// TwinCAT 3 PLC project PRG_MC_HMI_Conn
// Title: B_MachineControl_HMI_Connector
// Company: RafalOS
// Author: Rafal Osajda
// ProjectVersion: 0.0.0.38
// ProgramVersion: 3.1.4024.0
// libraries:
//   B_Base, * (RafalOS)
//   B_Base_HMI_Connector, * (RafalOS)
//   B_HMIElements, * (RafalOS)
//   B_MachineControl, * (RafalOS)
//   B_StatesAndModes, * (RafalOS)
//   VisuElemBase, * (System)
//   Tc2_Standard, * (Beckhoff Automation GmbH)
//   Tc2_System, * (Beckhoff Automation GmbH)
//   Tc3_Module, * (Beckhoff Automation GmbH)
//   VisuSymbols,3.5.10.0,System
// project tree:
//   DUTs/ ST_MCHMIPrepareScreen_List.TcDUT, ST_MCHMIPrepareScreen_DescriptorList.TcDUT
//   GVLs/ GVL_MCHMIConstans.TcGVL
//   / PlcTask.TcTTO (not stored)
//   POUs Compilation/ PRGCompilation.TcPOU
//   POUs/01_MC/ FB_MCHMIMachineControl_HMI.TcPOU, ITF_MCHMIMachineControl_HMI.TcIO, ITF_MCHMIMachineControl_HMI_PrepScr.TcIO, ITF_MCHMIMachineControl_HMI_PrepScr_00_01.TcIO, ITF_MCHMIMachineControl_HMI_PrepScr_00_02.TcIO, ITF_MCHMIMachineControl_HMI_PrepScr_00_03.TcIO, ITF_MCHMIMachineControl_HMI_PrepScr_00_04.TcIO, ITF_MCHMIMachineControl_HMI_PrepScr_00_05.TcIO, ITF_MCHMIMachineControl_HMI_PrepScr_01_XX.TcIO, ITF_MCHMIMachineControl_HMI_PrepScr_02_XX.TcIO, ITF_MCHMIMachineControl_HMI_PrepScr_03_XX.TcIO, ITF_MCHMIMachineControl_HMI_PrepScr_04_XX.TcIO, ITF_MCHMIMachineControl_HMI_PrepScr_05_XX.TcIO, ITF_MCHMIMachineControl_HMI_PrepScr_06_XX.TcIO, ITF_MCHMIMachineControl_HMI_PrepScr_07_XX.TcIO, ST_MCHMICommonData.TcDUT, ST_MCHMICommonData_RecipeInfo.TcDUT, ST_MCHMIMachineControl_HMI_Link.TcDUT, ST_MCHMIMachineControl_HMI.TcDUT
//   POUs/02_PrepareScreenParent/ FB_MCHMIPrepareDataForScreen.TcPOU, ITF_MCHMIDisplayExtension.TcIO, ITF_MCHMIPrepareDataForScreen.TcIO, ITF_MCHMIPrepareDataForScreenExtension.TcIO, ITF_MCHMIPrepareScreen_Init.TcIO
//   POUs/03_MW_Production/ FB_MCHMIPrepareDataForScreen_00_01.TcPOU, ITF_MCHMIPrepareScreen_00_01_Init.TcIO, ST_MCHMIPrepareScreen_00_01.TcDUT
//   POUs/04_MW_Maitenance/ FB_MCHMIPrepareDataForScreen_00_02.TcPOU, ITF_MCHMIPrepareScreen_00_02_Init.TcIO, ST_MCHMIPrepareScreen_00_02.TcDUT
//   POUs/05_MW_Manual/ FB_MCHMIPrepareDataForScreen_00_03.TcPOU, ITF_MCHMIPrepareScreen_00_03_Init.TcIO, ST_MCHMIPrepareScreen_00_03.TcDUT
//   POUs/06_MW_Washing/ FB_MCHMIPrepareDataForScreen_00_04.TcPOU, ITF_MCHMIPrepareScreen_00_04_Init.TcIO, ST_MCHMIPrepareScreen_00_04.TcDUT
//   POUs/07_MW_Diagnostics/ FB_MCHMIPrepareDataForScreen_00_05.TcPOU, ITF_MCHMIPrepareScreen_00_05_Init.TcIO, ST_MCHMIPrepareScreen_00_05.TcDUT
//   POUs/08_Parameters/ FB_MCHMIPrepareDataForScreen_01_XX.TcPOU, ITF_MCHMIPrepareScreen_01_XX_Init.TcIO, ST_MCHMIPrepareScreen_01_XX.TcDUT, ST_MCHMIPrepareScreen_01_XX_ElementList.TcDUT
//   POUs/09_Recipe/ FB_MCHMIPrepareDataForScreen_02_XX.TcPOU, ITF_MCHMIPrepareScreen_02_XX_Init.TcIO, ST_MCHMIPrepareScreen_02_XX.TcDUT, ST_MCHMIPrepareScreen_02_XX_AddRecipe.TcDUT, ST_MCHMIPrepareScreen_02_XX_DeleteRecipe.TcDUT
//   POUs/10_Alarm/ FB_MCHMIPrepareDataForScreen_03_XX.TcPOU, ITF_MCHMIPrepareScreen_03_XX_Init.TcIO, ST_MCHMIPrepareScreen_03_XX.TcDUT
//   POUs/11_ChangeMode/ FB_MCHMIPrepareDataForScreen_04_XX.TcPOU, ITF_MCHMIPrepareScreen_04_XX_Init.TcIO, ST_MCHMIPrepareScreen_04_XX.TcDUT
//   POUs/12_Statistics/ FB_MCHMIPrepareDataForScreen_05_XX.TcPOU, ITF_MCHMIPrepareScreen_05_XX_Init.TcIO, ST_MCHMIPrepareScreen_05_XX.TcDUT
//   POUs/13_StateDiagram/ FB_MCHMIPrepareDataForScreen_06_XX.TcPOU, ITF_MCHMIPrepareScreen_06_XX_Init.TcIO, ST_MCHMIPrepareScreen_06_XX.TcDUT, ST_MCHMIPrepareScreen_06_XX_ChangeMode.TcDUT, ST_MCHMIPrepareScreen_06_XX_CmdChangeState.TcDUT, ST_MCHMIPrepareScreen_06_XX_State.TcDUT
//   POUs/14_Setings/ FB_MCHMIPrepareDataForScreen_07_XX.TcPOU, ITF_MCHMIPrepareScreen_07_XX_Init.TcIO, ST_MCHMIPrepareScreen_07_XX.TcDUT
//   VISUs/ VisualizationManager.TcVMO (not stored)
// real-time tasks:
//   TASK PlcTask: cycle T#10ms, priority 20, ADS port 350

// ---- DUTs/ST_MCHMIPrepareScreen_List.TcDUT
TYPE ST_MCHMIPrepareScreen_List :
STRUCT
	arrRow					: ARRAY [1..GVL_MCHMIConstans.NUMBER_INDEGRIEND_ON_PAGE] OF ST_BaseHMIDescriptor;
	iSelectedRow			: INT; //numer wybranego składnika
	iSelectedRowPrev		: INT; //numer wybranego składnika - poprzedni
	bSelectedRow			: BOOL;
	
END_STRUCT
END_TYPE

// ---- DUTs/ST_MCHMIPrepareScreen_DescriptorList.TcDUT
TYPE ST_MCHMIPrepareScreen_DescriptorList :
STRUCT
	iTotal				: INT; //całkowita liczba danych do wyświetlenia
	iStartIndex			: INT; //liczba startowa
	iNumberRowOnPage	: INT; //liczbna wierszy na stronie
	iNumberOfPage		: INT; //ilosc stron potrzebnych do wyświetlenia wszystkich danych
	iActualPage			: INT; //aktualna strona
	iPreviewPage		: INT; //Poprzednia strona
	stChossenRow		: ST_BaseHMIDescriptorEdit;
	stList				: ST_MCHMIPrepareScreen_List;
	bRefresh			: BOOL;
END_STRUCT
END_TYPE

// ---- POUs/01_MC/ST_MCHMICommonData.TcDUT
TYPE ST_MCHMICommonData :
STRUCT
	bChangePage				: BOOL; //zmiana strony menu głównego
	wsActualState			: WSTRING;
	wsActualMode			: WSTRING;
	stRecipeInformation		: ST_MCHMICommonData_RecipeInfo;
END_STRUCT
END_TYPE

// ---- POUs/01_MC/ST_MCHMICommonData_RecipeInfo.TcDUT
TYPE ST_MCHMICommonData_RecipeInfo :
STRUCT
	bRecipeSelected			: BOOL;
	wsRecipeInformation		: WSTRING;
	dwBackgroud				: DWORD;
	dwText					: DWORD;
	(* rozpisane tło
	16#<TT><RR><GG><BB>
	<TT> 00-FF Transpoarency
	<RR> 00-FF red
	<GG> 00-FF green
	<BB> 00-FF blue
	*)
	bNewSelectedRecipe		: BOOL;
END_STRUCT
END_TYPE

// ---- POUs/01_MC/ST_MCHMIMachineControl_HMI_Link.TcDUT
TYPE ST_MCHMIMachineControl_HMI_Link EXTENDS ST_BaseTopElement_HMI_Link :
STRUCT
	stMachineControl		: ST_MCHMIMachineControl_HMI;
	stCommonData			: ST_MCHMICommonData;
	stPrepScr_00_01			: ST_MCHMIPrepareScreen_00_01;
	stPrepScr_00_02			: ST_MCHMIPrepareScreen_00_02;
	stPrepScr_00_03			: ST_MCHMIPrepareScreen_00_03;
	stPrepScr_00_04			: ST_MCHMIPrepareScreen_00_04;
	stPrepScr_00_05			: ST_MCHMIPrepareScreen_00_05;
	stPrepScr_01_XX			: ST_MCHMIPrepareScreen_01_XX;
	stPrepScr_02_XX			: ST_MCHMIPrepareScreen_02_XX;
	stPrepScr_03_XX			: ST_MCHMIPrepareScreen_03_XX;
	stPrepScr_04_XX			: ST_MCHMIPrepareScreen_04_XX;
	stPrepScr_05_XX			: ST_MCHMIPrepareScreen_05_XX;
	stPrepScr_06_XX			: ST_MCHMIPrepareScreen_06_XX;
	stPrepScr_07_XX			: ST_MCHMIPrepareScreen_07_XX;
	stRecipe				: ST_BaseRecipe_HMI;
END_STRUCT
END_TYPE

// ---- POUs/01_MC/ST_MCHMIMachineControl_HMI.TcDUT
TYPE ST_MCHMIMachineControl_HMI :
STRUCT
	bZmienna : BOOL;
END_STRUCT
END_TYPE

// ---- POUs/03_MW_Production/ST_MCHMIPrepareScreen_00_01.TcDUT
TYPE ST_MCHMIPrepareScreen_00_01 :
STRUCT
	btmpValue_00_01	: BOOL;
END_STRUCT
END_TYPE

// ---- POUs/04_MW_Maitenance/ST_MCHMIPrepareScreen_00_02.TcDUT
TYPE ST_MCHMIPrepareScreen_00_02 :
STRUCT
	btmpValue_00_02	: BOOL;
END_STRUCT
END_TYPE

// ---- POUs/05_MW_Manual/ST_MCHMIPrepareScreen_00_03.TcDUT
TYPE ST_MCHMIPrepareScreen_00_03 :
STRUCT
	btmpValue_00_03	: BOOL;
END_STRUCT
END_TYPE

// ---- POUs/06_MW_Washing/ST_MCHMIPrepareScreen_00_04.TcDUT
TYPE ST_MCHMIPrepareScreen_00_04 :
STRUCT
	btmpValue_00_04	: BOOL;
END_STRUCT
END_TYPE

// ---- POUs/07_MW_Diagnostics/ST_MCHMIPrepareScreen_00_05.TcDUT
TYPE ST_MCHMIPrepareScreen_00_05 :
STRUCT
	btmpValue_00_05	: BOOL;
END_STRUCT
END_TYPE

// ---- POUs/08_Parameters/ST_MCHMIPrepareScreen_01_XX.TcDUT
TYPE ST_MCHMIPrepareScreen_01_XX :
STRUCT
	stListElement			: ST_MCHMIPrepareScreen_01_XX_ElementList;
	
END_STRUCT
END_TYPE

// ---- POUs/08_Parameters/ST_MCHMIPrepareScreen_01_XX_ElementList.TcDUT
TYPE ST_MCHMIPrepareScreen_01_XX_ElementList :
STRUCT
	arrNames 			: ARRAY  [1..GVL_BaseConstans.MAX_NUMBER_OF_ALL_ITEM] OF WSTRING;
	arrID				: ARRAY  [1..GVL_BaseConstans.MAX_NUMBER_OF_ALL_ITEM] OF UINT;
	iNumber				: INT;	//liczba elementów z parametrami
	itfElement			: ITF_BaseComponent_HMI;	//interfejs wybranego elementu
END_STRUCT
END_TYPE

// ---- POUs/09_Recipe/ST_MCHMIPrepareScreen_02_XX.TcDUT
TYPE ST_MCHMIPrepareScreen_02_XX :
STRUCT
	bRefreshList		: BOOL;	//odświerzenie listy po zmianie listy receptur
	arrNameListRecipe	: ARRAY [1..GVL_BaseConstans.MAX_NUMBER_OF_RECIPES] OF WSTRING;
	arrNameListTemplate	: ARRAY [1..GVL_BaseConstans.MAX_NUMBER_OF_RECIPES] OF WSTRING;
	iNumberOfRecipe		: INT;
	iNumberOfTemplate	: INT;
	iSelectedNameRow	: INT;
	iSelectedNameRowPrev 	: INT; //poprzedni wiersz listy receptur
	bSelectedNameRow	: BOOL;
(*	Wyświetlanie składników	*)
	stIngredientList	: ST_MCHMIPrepareScreen_DescriptorList;
	
(*	Widoczność przycisków	*)
	bVisibleButtonAddFromTemplate	: BOOL;
	bVisibleButtonAddFromRecipe		: BOOL;
	bVisibleButtonDelete			: BOOL;
	bVsibleButtonEditIngredient		: BOOL;
	bVisibleButtonChoose			: BOOL;
	
(*	Tworzenie nowej receptury	- ramka	*)
	stAddRecipe			: ST_MCHMIPrepareScreen_02_XX_AddRecipe;
(*	Ususwanie receptury	*)
	stDeleteRecipe		: ST_MCHMIPrepareScreen_02_XX_DeleteRecipe;
(*	Wybieranie receptury	*)
	bSelectRecipe		: BOOL;
	
END_STRUCT
END_TYPE

// ---- POUs/09_Recipe/ST_MCHMIPrepareScreen_02_XX_AddRecipe.TcDUT
TYPE ST_MCHMIPrepareScreen_02_XX_AddRecipe :
STRUCT
	bNewRecipeFromTemplate	: BOOL;
	bNewRecipeFromRecipe	: BOOL;
	arrListOfName			: ARRAY [1..GVL_BaseConstans.MAX_NUMBER_OF_RECIPES ] OF WSTRING;
	iNumberOfNames			: INT;
	iSelectedName			: INT;
	bSelectedRow			: BOOL;
	stNewNames				: ST_BaseLabel;	//nazwa nowej receptury
	bOk						: BOOL;
	bCancel					: BOOL;	
	wsTitle					: WSTRING;
	wsSource				: WSTRING;
END_STRUCT
END_TYPE

// ---- POUs/09_Recipe/ST_MCHMIPrepareScreen_02_XX_DeleteRecipe.TcDUT
TYPE ST_MCHMIPrepareScreen_02_XX_DeleteRecipe :
STRUCT
	bDeleteRecipe		: BOOL;
	bOK					: BOOL;
	bCancel				: BOOL;
	wsDescription		: WSTRING;
	wsNameRecipe		: WSTRING;
	
END_STRUCT
END_TYPE

// ---- POUs/10_Alarm/ST_MCHMIPrepareScreen_03_XX.TcDUT
TYPE ST_MCHMIPrepareScreen_03_XX :
STRUCT
	btmpValue_03_XX	: BOOL;
END_STRUCT
END_TYPE

// ---- POUs/11_ChangeMode/ST_MCHMIPrepareScreen_04_XX.TcDUT
TYPE ST_MCHMIPrepareScreen_04_XX :
STRUCT
	wsActualMode			: WSTRING;
	eActualMode				: E_BaseMachineMode;
	
	bChangeMode				: BOOL;	//zmien tryb polecenie z HMi
	iSelectedMode			: INT;
	iNumberModeToDisplay	: INT;
	arrNamesOfMode			: ARRAY [0..GVL_SaMConstans.NUMBER_OF_MODES] OF ST_MCHMIPrepareScreen_06_XX_ChangeMode;
	bSelectedRow			: BOOL;
END_STRUCT
END_TYPE

// ---- POUs/12_Statistics/ST_MCHMIPrepareScreen_05_XX.TcDUT
TYPE ST_MCHMIPrepareScreen_05_XX :
STRUCT
	btmpValue_05_XX	: BOOL;
END_STRUCT
END_TYPE

// ---- POUs/13_StateDiagram/ST_MCHMIPrepareScreen_06_XX.TcDUT
TYPE ST_MCHMIPrepareScreen_06_XX :
STRUCT
	wsActualState			: WSTRING;
	wsActualMode			: WSTRING;
	eActualMode				: E_BaseMachineMode;
	(*	Informacje o stanach w trybie	*)
	arrState				: ARRAY [0..GVL_SaMConstans.NUMBER_OF_STATES] OF ST_MCHMIPrepareScreen_06_XX_State;
	arrStateEnabledInMode	: ARRAY [0..GVL_SaMConstans.NUMBER_OF_STATES] OF BOOL;
	(*	Dane dotyczące wyświetlania czasów 	*)
	bShowTime				: BOOL;
	sTotalWorkTime			: STRING;
	iNumberModeToShowTime	: INT;
	sWorkingTimeInMode		: STRING;
	sNameOfModeShown		: STRING;	//nazwa trybu pokazywanego trybu
	bNextModeToDisplayTime	: BOOL;
	bPrevModeToDisplayTime	: BOOL;
	wsNameModeOfTimeDisplay	: WSTRING;

	
	(*	Przyciski poleceń zmiany stany	*)
	arrCmdChangeState		: ARRAY [1..GVL_SaMConstans.NUMBER_OF_COMMAND_CHANGE_STATES] OF ST_MCHMIPrepareScreen_06_XX_CmdChangeState;

	(*	Obsługa zmiany trybu	*)
	bChangeMode				: BOOL;	//zmien tryb polecenie z HMi
	iSelectedMode			: INT;
	iNumberModeToDisplay	: INT;
	arrNamesOfMode			: ARRAY [0..GVL_SaMConstans.NUMBER_OF_MODES] OF ST_MCHMIPrepareScreen_06_XX_ChangeMode;
	bSelectedRow			: BOOL;
END_STRUCT
END_TYPE

// ---- POUs/13_StateDiagram/ST_MCHMIPrepareScreen_06_XX_ChangeMode.TcDUT
TYPE ST_MCHMIPrepareScreen_06_XX_ChangeMode :
STRUCT
	wsDescription			: WSTRING;
	iNumber					: INT;	//numer trybu
END_STRUCT
END_TYPE

// ---- POUs/13_StateDiagram/ST_MCHMIPrepareScreen_06_XX_CmdChangeState.TcDUT
TYPE ST_MCHMIPrepareScreen_06_XX_CmdChangeState :
STRUCT
	bPushed		: BOOL;
	bEnabled	: BOOL;
END_STRUCT
END_TYPE

// ---- POUs/13_StateDiagram/ST_MCHMIPrepareScreen_06_XX_State.TcDUT
TYPE ST_MCHMIPrepareScreen_06_XX_State :
STRUCT
	wsNameOfState			: WSTRING;
	iWidthFrame				: INT := 1;
	bShowTime				: BOOL;
	sTime					: STRING;
	dwBackgroud				: DWORD;
	(* rozpisane tło
	16#<TT><RR><GG><BB>
	<TT> 00-FF Transpoarency
	<RR> 00-FF red
	<GG> 00-FF green
	<BB> 00-FF blue
	*)
END_STRUCT
END_TYPE

// ---- POUs/14_Setings/ST_MCHMIPrepareScreen_07_XX.TcDUT
TYPE ST_MCHMIPrepareScreen_07_XX :
STRUCT
	arrLocationDescription	: ARRAY  [0..GVL_BaseConstans.NUMBER_OF_LOCATIONS] OF WSTRING;
	iChoosoLocation			: INT;
	
	bCreateRecipeTemplate 	: BOOL;
END_STRUCT
END_TYPE

// ---- GVLs/GVL_MCHMIConstans.TcGVL
{attribute 'qualified_only'}
VAR_GLOBAL CONSTANT
	NUMBER_INDEGRIEND_ON_PAGE	: INT := 10;	//liczba wyświetlanych składników recepury w trybie domyślnym
	
END_VAR

// ---- POUs/01_MC/ITF_MCHMIMachineControl_HMI.TcIO
(*			
	RafalOS
	Rafał Osajda		20.11.2025		TC 4024.66
	Interfejs umożliwający wywoływanie moted z HMIManager
*)
INTERFACE ITF_MCHMIMachineControl_HMI EXTENDS ITF_BaseTopElement_HMI

METHOD PUBLIC AddPrepareScreenModuleFromManager : BOOL
VAR_INPUT
	itfModule	: ITF_MCHMIPrepareScreen_Init;// ITF_MCHMIPrepareDataForScreen;
END_VAR
END_METHOD

(*			
	RafalOS
	Rafał Osajda		26.11.2025		TC 4024.66
	Podłaczenie modułu receptur
*)
METHOD PUBLIC AddRecipeModulFormManager : BOOL
VAR_INPUT
	fbRecipeModul		: ITF_BaseRecipe_HMI;
END_VAR
END_METHOD

(*			
	RafalOS
	Rafał Osajda		19.11.2025		TC 4024.66
	Sprzątanie po stronie wywoływane z HMIManager i wywołująca odpowiednią metode z ITF z arrPrepareScreen
*)
METHOD ClearAfterScreenFroHMIManager : BOOL
VAR_INPUT
	iScreen		: INT;
	iMode		: INT;
END_VAR
END_METHOD

METHOD PUBLIC GetActiveModeFromManager : E_BaseMachineMode
VAR_INPUT
END_VAR
END_METHOD

(*			
	RafalOS
	Rafał Osajda		07.12.2025		TC 4024.66
	Pobierz informacje o aktualnym stanie recepur tzn o tym czy jest wybrana a jak tak to która
*)
METHOD PUBLIC GetInformationLatestRecipes
VAR_INPUT
END_VAR
END_METHOD

METHOD PUBLIC LinkMachineControlData : BOOL
VAR_INPUT
	stData			: REFERENCE TO ST_MCHMIMachineControl_HMI_Link;
END_VAR
END_METHOD

(*			
	RafalOS
	Rafał Osajda		20.11.2025		TC 4024.66
	Podpięcie modułu generowania danych do odpowiedniej pozycji w tablicy [Okno][Tryb]
*)
METHOD PUBLIC LinkPrepareScreenToArrayFromConfiguration : BOOL
VAR_INPUT
	iScreen		: INT;
	iMode		: INT;
	itfModule	: ITF_MCHMIPrepareDataForScreen;
END_VAR
END_METHOD

(*			
	RafalOS
	Rafał Osajda		19.11.2025		TC 4024.66
	Przygotowanie danych dla strony wywoływane z HMIManager i wywołująca odpowiednią metode z ITF z arrPrepareScreen
*)
METHOD PrepareDataForScreenFromHMIManager : BOOL
VAR_INPUT
	iScreen		: INT;
	iMode		: INT;
END_VAR
END_METHOD

(*			
	RafalOS
	Rafał Osajda		19.11.2025		TC 4024.66
	Przygotowanie strony wywoływane z HMIManager i wywołująca odpowiednią metode z ITF z arrPrepareScreen
*)
METHOD PrepareForScreenFromHMIManager : BOOL
VAR_INPUT
	iScreen		: INT;
	iMode		: INT;
END_VAR
END_METHOD

(*			
	RafalOS
	Rafał Osajda		20.11.2025		TC 4024.66
	Ustawienei zmiennej w wspólnych zmiennych z managera
*)
METHOD PUBLIC SetChangePageFromManager : BOOL
VAR_INPUT
	bValue	: BOOL;
END_VAR
END_METHOD

END_INTERFACE

// ---- POUs/01_MC/ITF_MCHMIMachineControl_HMI_PrepScr.TcIO
INTERFACE ITF_MCHMIMachineControl_HMI_PrepScr EXTENDS ITF_MCHMIMachineControl_HMI_PrepScr_00_01, 
	ITF_MCHMIMachineControl_HMI_PrepScr_00_02,
	ITF_MCHMIMachineControl_HMI_PrepScr_00_03,
	ITF_MCHMIMachineControl_HMI_PrepScr_00_04,
	ITF_MCHMIMachineControl_HMI_PrepScr_00_05,
	ITF_MCHMIMachineControl_HMI_PrepScr_01_XX,
	ITF_MCHMIMachineControl_HMI_PrepScr_02_XX,
	ITF_MCHMIMachineControl_HMI_PrepScr_03_XX,
	ITF_MCHMIMachineControl_HMI_PrepScr_04_XX,
	ITF_MCHMIMachineControl_HMI_PrepScr_05_XX,
	ITF_MCHMIMachineControl_HMI_PrepScr_06_XX,
	ITF_MCHMIMachineControl_HMI_PrepScr_07_XX

END_INTERFACE

// ---- POUs/01_MC/ITF_MCHMIMachineControl_HMI_PrepScr_00_01.TcIO
(*			
	RafalOS
	Rafał Osajda		20.11.2025		TC 4024.66
	Interfejs przekazywany do modułów tworzących strony
*)
INTERFACE ITF_MCHMIMachineControl_HMI_PrepScr_00_01

END_INTERFACE

// ---- POUs/01_MC/ITF_MCHMIMachineControl_HMI_PrepScr_00_02.TcIO
(*			
	RafalOS
	Rafał Osajda		20.11.2025		TC 4024.66
	Interfejs przekazywany do modułów tworzących strony
*)
INTERFACE ITF_MCHMIMachineControl_HMI_PrepScr_00_02

END_INTERFACE

// ---- POUs/01_MC/ITF_MCHMIMachineControl_HMI_PrepScr_00_03.TcIO
(*			
	RafalOS
	Rafał Osajda		20.11.2025		TC 4024.66
	Interfejs przekazywany do modułów tworzących strony
*)
INTERFACE ITF_MCHMIMachineControl_HMI_PrepScr_00_03

END_INTERFACE

// ---- POUs/01_MC/ITF_MCHMIMachineControl_HMI_PrepScr_00_04.TcIO
(*			
	RafalOS
	Rafał Osajda		20.11.2025		TC 4024.66
	Interfejs przekazywany do modułów tworzących strony
*)
INTERFACE ITF_MCHMIMachineControl_HMI_PrepScr_00_04

END_INTERFACE

// ---- POUs/01_MC/ITF_MCHMIMachineControl_HMI_PrepScr_00_05.TcIO
(*			
	RafalOS
	Rafał Osajda		20.11.2025		TC 4024.66
	Interfejs przekazywany do modułów tworzących strony
*)
INTERFACE ITF_MCHMIMachineControl_HMI_PrepScr_00_05

END_INTERFACE

// ---- POUs/01_MC/ITF_MCHMIMachineControl_HMI_PrepScr_01_XX.TcIO
(*			
	RafalOS
	Rafał Osajda		20.11.2025		TC 4024.66
	Interfejs przekazywany do modułów tworzących strony
*)
INTERFACE ITF_MCHMIMachineControl_HMI_PrepScr_01_XX

(*			
	RafalOS
	Rafał Osajda		17.12.2025		TC 4024.66
	Pobiera listę elementów które posiadaja parametr i 
	przypisuje ja do zadanej struktury i zwraca true jak się uda
*)
METHOD GetElementNamesWithParameter : BOOL
VAR_INPUT
	stDane			: REFERENCE TO ST_MCElementListWithParameter;
END_VAR
END_METHOD

END_INTERFACE

// ---- POUs/01_MC/ITF_MCHMIMachineControl_HMI_PrepScr_02_XX.TcIO
(*			
	RafalOS
	Rafał Osajda		20.11.2025		TC 4024.66
	Interfejs przekazywany do modułów tworzących strony
*)
INTERFACE ITF_MCHMIMachineControl_HMI_PrepScr_02_XX

(*			
	RafalOS
	Rafał Osajda		03.03.2025		TC 4026.13		wer. 0.0.0.1
	Kopiuje składniki z wybranej receptury i tworzy nową recepture
*)
METHOD PUBLIC AddRecipeFromRecipe : BOOL
VAR_INPUT
	uiNumberRecipe				: UINT;
	stTexts						: ST_BaseLabel;
END_VAR
END_METHOD

(*			
	RafalOS
	Rafał Osajda		03.03.2025		TC 4026.13		wer. 0.0.0.1
	Kopiuje składniki z wybranego szablonu i tworzy nową recepture
*)
METHOD PUBLIC AddRecipeFromTemplate : BOOL
VAR_INPUT
	uiNumberTemplates			: UINT;
	stTexts						: ST_BaseLabel;
END_VAR
END_METHOD

(*			
	RafalOS
	Rafał Osajda		03.06.2025		TC 4024.66
	usuwa referencje do wybranej
*)
METHOD PUBLIC ClearChosen
VAR_INPUT
END_VAR
END_METHOD

(*			
	RafalOS
	Rafał Osajda		03.03.2025		TC 4026.13		wer. 0.0.0.1
	
*)
METHOD PUBLIC DeleteRecipe : BOOL
VAR_INPUT
	uiNumber				: uint;
END_VAR
END_METHOD

(*			
	RafalOS
	Rafał Osajda		03.03.2025		TC 4026.13		wer. 0.0.0.1
	
*)
METHOD PUBLIC GetIngredientFromRecipe : ST_BaseDescriptor
VAR_INPUT
	uiNumberOfRecipe			: UINT;
	uiNumberOfIngredient		: UINT;
END_VAR
END_METHOD

(*			
	RafalOS
	Rafał Osajda		02.12.2025		TC 4024.66
	Zwraca do tablicy wybrany zakres składników
*)
METHOD PUBLIC GetIngredientRange 
VAR_INPUT
	iRecipe			: INT;	//numer receptury z której bierzemy składniki
	iStartIndex		: INT;	//numer startowy składnika
	iCount			: INT;	//ilośc pobieranych 
END_VAR
VAR_IN_OUT
	arrOut : ARRAY [*] OF ST_BaseDescriptor;
END_VAR
VAR_OUTPUT
	iNumberOfFilledData	: INT;	//ilosc wypelnionych danych na strone
END_VAR
END_METHOD

METHOD PUBLIC GetListOfNameRecipe : ST_BaseRecipeList
VAR_INPUT
END_VAR
END_METHOD

METHOD PUBLIC GetListOfNameTemplate : ST_BaseRecipeList
VAR_INPUT
END_VAR
END_METHOD

(*			
	RafalOS
	Rafał Osajda		03.03.2025		TC 4026.13		wer. 0.0.0.1
	
*)
METHOD PUBLIC GetNumberIngredientOfRecipe : UINT
VAR_INPUT
	uiNumber				: UINT;
END_VAR
END_METHOD

METHOD PUBLIC GetNumberOfChoosen : UINT
VAR_INPUT
END_VAR
END_METHOD

METHOD PUBLIC GetNumberOfRecipe : UINT
VAR_INPUT
END_VAR
END_METHOD

METHOD PUBLIC GetNumberOfTemplate : UINT
VAR_INPUT
END_VAR
END_METHOD

(*			
	RafalOS
	Rafał Osajda		06.12.2025		TC 4024.66
	Wybranie receputury
*)
METHOD SelectRecipe : BOOL
VAR_INPUT
	uiRecipe: UINT;
END_VAR
END_METHOD

(*			
	RafalOS
	Rafał Osajda		05.12.2025		TC 4024.66
	Ustawia nową wartośc w podanym składniku
*)
METHOD PUBLIC SetIngredientValue
VAR_INPUT
	iRecipe			: int;
	iIngredient		: INT;
	rValue			: REAL;
END_VAR
END_METHOD

END_INTERFACE

// ---- POUs/01_MC/ITF_MCHMIMachineControl_HMI_PrepScr_03_XX.TcIO
(*			
	RafalOS
	Rafał Osajda		20.11.2025		TC 4024.66
	Interfejs przekazywany do modułów tworzących strony
*)
INTERFACE ITF_MCHMIMachineControl_HMI_PrepScr_03_XX

END_INTERFACE

// ---- POUs/01_MC/ITF_MCHMIMachineControl_HMI_PrepScr_04_XX.TcIO
(*			
	RafalOS
	Rafał Osajda		20.11.2025		TC 4024.66
	Interfejs przekazywany do modułów tworzących strony
*)
INTERFACE ITF_MCHMIMachineControl_HMI_PrepScr_04_XX

METHOD GetActiveMode : E_BaseMachineMode
VAR_INPUT
END_VAR
END_METHOD

METHOD PUBLIC GetActiveModeName : ST_BaseLabel
VAR_INPUT
END_VAR
END_METHOD

(*			
	RafalOS
	Rafał Osajda		25.11.2025		TC 4024.66
	Zwraca nazwę trybu o zadanym numerze
*)
METHOD GetModeName : ST_BaseLabel
VAR_INPUT
	iMode	: INT;
END_VAR
END_METHOD

(*			
	RafalOS
	Rafał Osajda		25.11.2025		TC 4024.66
	Zwraca czy tryb o podanym numerze jest włączony
*)
METHOD IsModeEnabled : BOOL
VAR_INPUT
	iMode 	: INT;
END_VAR
END_METHOD

(*			
	RafalOS
	Rafał Osajda		24.11.2025		TC 4024.66
	Zmien tryb
*)
METHOD SetCmdChangeMode : BOOL
VAR_INPUT
	eCmdNumber	: E_SaMCommandChangeMode;
END_VAR
END_METHOD

END_INTERFACE

// ---- POUs/01_MC/ITF_MCHMIMachineControl_HMI_PrepScr_05_XX.TcIO
(*			
	RafalOS
	Rafał Osajda		20.11.2025		TC 4024.66
	Interfejs przekazywany do modułów tworzących strony
*)
INTERFACE ITF_MCHMIMachineControl_HMI_PrepScr_05_XX

END_INTERFACE

// ---- POUs/01_MC/ITF_MCHMIMachineControl_HMI_PrepScr_06_XX.TcIO
(*			
	RafalOS
	Rafał Osajda		20.11.2025		TC 4024.66
	Interfejs przekazywany do modułów tworzących strony
*)
INTERFACE ITF_MCHMIMachineControl_HMI_PrepScr_06_XX

METHOD GetActiveMode : E_BaseMachineMode
VAR_INPUT
END_VAR
END_METHOD

METHOD PUBLIC GetActiveModeName : ST_BaseLabel
VAR_INPUT
END_VAR
END_METHOD

METHOD GetActiveState : E_BaseMachineState
VAR_INPUT
END_VAR
END_METHOD

METHOD PUBLIC GetActiveStateName : ST_BaseLabel
VAR_INPUT
END_VAR
END_METHOD

(*			
	RafalOS
	Rafał Osajda		25.11.2025		TC 4024.66
	Zwraca nazwę trybu o zadanym numerze
*)
METHOD GetModeName : ST_BaseLabel
VAR_INPUT
	iMode	: INT;
END_VAR
END_METHOD

METHOD GetStateName : ST_BaseLabel
VAR_INPUT
	iNumber		: INT;
END_VAR
END_METHOD

METHOD GetStateTimeForMode : LTIME
VAR_INPUT
	iMode		: INT;
	iState		: INT;
END_VAR
END_METHOD

METHOD GetTimeWorkForMode : LTIME
VAR_INPUT
	iMode	: INT;
END_VAR
END_METHOD

(*			
	RafalOS
	Rafał Osajda		25.11.2025		TC 4024.66
	Zwraca całkowity czas pracy maszyny
*)
METHOD PUBLIC GetTotalWorkTime : LTIME
VAR_INPUT
END_VAR
END_METHOD

(*			
	RafalOS
	Rafał Osajda		25.11.2025		TC 4024.66
	Zwraca czy zmiana stanu sie skońćzyła
*)
METHOD IsChangeModeDone : BOOL
VAR_INPUT
END_VAR
END_METHOD

(*			
	RafalOS
	Rafał Osajda		25.11.2025		TC 4024.66
	Zwraca czy tryb o podanym numerze jest włączony
*)
METHOD IsModeEnabled : BOOL
VAR_INPUT
	iMode 	: INT;
END_VAR
END_METHOD

METHOD IsStateActive : BOOL
VAR_INPUT
	iTestState : INT;
END_VAR
END_METHOD

METHOD IsStateEnableInMode : BOOL
VAR_INPUT
	iTestState	: INT;
END_VAR
END_METHOD

(*			
	RafalOS
	Rafał Osajda		24.11.2025		TC 4024.66
	Zmien tryb
*)
METHOD SetCmdChangeMode : BOOL
VAR_INPUT
	eCmdNumber	: E_SaMCommandChangeMode;
END_VAR
END_METHOD

(*			
	RafalOS
	Rafał Osajda		24.11.2025		TC 4024.66
	Zmien stan 
*)
METHOD public SetCmdChangeState : BOOL
VAR_INPUT
	eCmdNumber : E_SaMCommandChangeState;
END_VAR
END_METHOD

END_INTERFACE

// ---- POUs/01_MC/ITF_MCHMIMachineControl_HMI_PrepScr_07_XX.TcIO
(*			
	RafalOS
	Rafał Osajda		20.11.2025		TC 4024.66
	Interfejs przekazywany do modułów tworzących strony
*)
INTERFACE ITF_MCHMIMachineControl_HMI_PrepScr_07_XX

(*			
	RafalOS
	Rafał Osajda		25.10.2025		TC 4024.66
	Utworzenie nowych szablonów receptur na podstawie dodanych fb zewnętrznych - wywołanie metody powoduje
	skosowanie dotychczasowych szablonów i receptur
*)
METHOD PUBLIC CreateRecipeTemplates : BOOL
VAR_INPUT
END_VAR
END_METHOD

END_INTERFACE

// ---- POUs/02_PrepareScreenParent/ITF_MCHMIDisplayExtension.TcIO
INTERFACE ITF_MCHMIDisplayExtension

(*			
	RafalOS
	Rafał Osajda		19.11.2025		TC 4024.66
	Czyści danych przy zmienia ramki po poprzedniej ramce
*)
METHOD PUBLIC ExtendedClearAfterScreen : BOOL
VAR_INPUT
END_VAR
END_METHOD

(*			
	RafalOS
	Rafał Osajda		20.11.2025		TC 4024.66
	Przygotuj rozszerzone wyświetlanie
*)
METHOD PUBLIC ExtendedPrepareDataForHMI : BOOL
VAR_INPUT
END_VAR
END_METHOD

(*			
	RafalOS
	Rafał Osajda		19.11.2025		TC 4024.66
	Przygotowanie ramki pood tamke do wyświetlenia - tylko przygotowanie a nie przygotowanie danych do wyświetlenia
*)
METHOD PUBLIC ExtendedPrepareForScreen : BOOL
VAR_INPUT
END_VAR
END_METHOD

END_INTERFACE

// ---- POUs/02_PrepareScreenParent/ITF_MCHMIPrepareDataForScreen.TcIO
INTERFACE ITF_MCHMIPrepareDataForScreen EXTENDS ITF_BaseComponent_HMI

(*			
	RafalOS
	Rafał Osajda		19.11.2025		TC 4024.66
	Czyści danych przy zmienia ramki po poprzedniej ramce
*)
METHOD PUBLIC ClearAfterScreen : BOOL
VAR_INPUT
END_VAR
END_METHOD

(*			
	RafalOS
	Rafał Osajda		14.11.2025		TC 4024.66
	Metoda przygotowywania danych dla HMI 
	W niej odbywa się odpytywanie właściego elementu przez łącznik
*)
METHOD PUBLIC PrepareDataForHMI : BOOL
VAR_INPUT
END_VAR
END_METHOD

(*			
	RafalOS
	Rafał Osajda		19.11.2025		TC 4024.66
	Przygotowanie ramki pood tamke do wyświetlenia - tylko przygotowanie a nie przygotowanie danych do wyświetlenia
*)
METHOD PUBLIC PrepareForScreen : BOOL
VAR_INPUT
END_VAR
END_METHOD

END_INTERFACE

// ---- POUs/02_PrepareScreenParent/ITF_MCHMIPrepareDataForScreenExtension.TcIO
INTERFACE ITF_MCHMIPrepareDataForScreenExtension

METHOD PUBLIC LinkExtensionDisplay : BOOL
VAR_INPUT
	fbExtendedDisplay			: ITF_MCHMIDisplayExtension;
END_VAR
END_METHOD

END_INTERFACE

// ---- POUs/02_PrepareScreenParent/ITF_MCHMIPrepareScreen_Init.TcIO
INTERFACE ITF_MCHMIPrepareScreen_Init EXTENDS ITF_MCHMIPrepareDataForScreen,
	ITF_MCHMIPrepareScreen_00_01_Init, 
	ITF_MCHMIPrepareScreen_00_02_Init,
	ITF_MCHMIPrepareScreen_00_03_Init,
	ITF_MCHMIPrepareScreen_00_04_Init,
	ITF_MCHMIPrepareScreen_00_05_Init,
	ITF_MCHMIPrepareScreen_01_XX_Init,
	ITF_MCHMIPrepareScreen_02_XX_Init,
	ITF_MCHMIPrepareScreen_03_XX_Init,
	ITF_MCHMIPrepareScreen_04_XX_Init,
	ITF_MCHMIPrepareScreen_05_XX_Init,
	ITF_MCHMIPrepareScreen_06_XX_Init,
	ITF_MCHMIPrepareScreen_07_XX_Init,
	ITF_MCHMIPrepareDataForScreenExtension

(*			
	RafalOS
	Rafał Osajda		20.11.2025		TC 4024.66
	Podłączenie wspólnych danych do modułu 
*)
METHOD PUBLIC LinkHMICommonData : BOOL
VAR_INPUT
	stHMICommonData	: REFERENCE TO ST_MCHMICommonData;
END_VAR
END_METHOD

END_INTERFACE

// ---- POUs/03_MW_Production/ITF_MCHMIPrepareScreen_00_01_Init.TcIO
INTERFACE ITF_MCHMIPrepareScreen_00_01_Init

METHOD PUBLIC LinkDataHMI_00_01 : BOOL
VAR_INPUT
	refstData				: REFERENCE TO ST_MCHMIPrepareScreen_00_01;
END_VAR
END_METHOD

END_INTERFACE

// ---- POUs/04_MW_Maitenance/ITF_MCHMIPrepareScreen_00_02_Init.TcIO
INTERFACE ITF_MCHMIPrepareScreen_00_02_Init

METHOD PUBLIC LinkDataHMI_00_02 : BOOL
VAR_INPUT
	refstData				: REFERENCE TO ST_MCHMIPrepareScreen_00_02;
END_VAR
END_METHOD

END_INTERFACE

// ---- POUs/05_MW_Manual/ITF_MCHMIPrepareScreen_00_03_Init.TcIO
INTERFACE ITF_MCHMIPrepareScreen_00_03_Init

METHOD PUBLIC LinkDataHMI_00_03 : BOOL
VAR_INPUT
	refstData				: REFERENCE TO ST_MCHMIPrepareScreen_00_03;
END_VAR
END_METHOD

END_INTERFACE

// ---- POUs/06_MW_Washing/ITF_MCHMIPrepareScreen_00_04_Init.TcIO
INTERFACE ITF_MCHMIPrepareScreen_00_04_Init

METHOD PUBLIC LinkDataHMI_00_04 : BOOL
VAR_INPUT
	refstData				: REFERENCE TO ST_MCHMIPrepareScreen_00_04;
END_VAR
END_METHOD

END_INTERFACE

// ---- POUs/07_MW_Diagnostics/ITF_MCHMIPrepareScreen_00_05_Init.TcIO
INTERFACE ITF_MCHMIPrepareScreen_00_05_Init

METHOD PUBLIC LinkDataHMI_00_05 : BOOL
VAR_INPUT
	refstData				: REFERENCE TO ST_MCHMIPrepareScreen_00_05;
END_VAR
END_METHOD

END_INTERFACE

// ---- POUs/08_Parameters/ITF_MCHMIPrepareScreen_01_XX_Init.TcIO
INTERFACE ITF_MCHMIPrepareScreen_01_XX_Init

METHOD PUBLIC LinkDataHMI_01_XX : BOOL
VAR_INPUT
	refstData				: REFERENCE TO ST_MCHMIPrepareScreen_01_XX;
END_VAR
END_METHOD

END_INTERFACE

// ---- POUs/09_Recipe/ITF_MCHMIPrepareScreen_02_XX_Init.TcIO
INTERFACE ITF_MCHMIPrepareScreen_02_XX_Init

METHOD PUBLIC LinkDataHMI_02_XX : BOOL
VAR_INPUT
	refstData				: REFERENCE TO ST_MCHMIPrepareScreen_02_XX;
END_VAR
END_METHOD

END_INTERFACE

// ---- POUs/10_Alarm/ITF_MCHMIPrepareScreen_03_XX_Init.TcIO
INTERFACE ITF_MCHMIPrepareScreen_03_XX_Init

METHOD PUBLIC LinkDataHMI_03_XX : BOOL
VAR_INPUT
	refstData				: REFERENCE TO ST_MCHMIPrepareScreen_03_XX;
END_VAR
END_METHOD

END_INTERFACE

// ---- POUs/11_ChangeMode/ITF_MCHMIPrepareScreen_04_XX_Init.TcIO
INTERFACE ITF_MCHMIPrepareScreen_04_XX_Init

METHOD PUBLIC LinkDataHMI_04_XX : BOOL
VAR_INPUT
	refstData				: REFERENCE TO ST_MCHMIPrepareScreen_04_XX;
END_VAR
END_METHOD

END_INTERFACE

// ---- POUs/12_Statistics/ITF_MCHMIPrepareScreen_05_XX_Init.TcIO
INTERFACE ITF_MCHMIPrepareScreen_05_XX_Init

METHOD PUBLIC LinkDataHMI_05_XX : BOOL
VAR_INPUT
	refstData				: REFERENCE TO ST_MCHMIPrepareScreen_05_XX;
END_VAR
END_METHOD

END_INTERFACE

// ---- POUs/13_StateDiagram/ITF_MCHMIPrepareScreen_06_XX_Init.TcIO
INTERFACE ITF_MCHMIPrepareScreen_06_XX_Init

METHOD PUBLIC LinkDataHMI_06_XX : BOOL
VAR_INPUT
	refstData				: REFERENCE TO ST_MCHMIPrepareScreen_06_XX;
END_VAR
END_METHOD

END_INTERFACE

// ---- POUs/14_Setings/ITF_MCHMIPrepareScreen_07_XX_Init.TcIO
INTERFACE ITF_MCHMIPrepareScreen_07_XX_Init

METHOD PUBLIC LinkDataHMI_07_XX : BOOL
VAR_INPUT
	refstData				: REFERENCE TO ST_MCHMIPrepareScreen_07_XX;
END_VAR
END_METHOD

END_INTERFACE

// ---- POUs Compilation/PRGCompilation.TcPOU
PROGRAM PRGCompilation
VAR
	fbLogger						: FB_BaseLogger;
	fbMachineControl				: FB_MCMachineControl;
	fbMachineControlHMIConnector	: FB_MCHMIMachineControl_HMI (
										itfBaseLoggerConnector		:= fbLogger,
	                                    itfMachineControlConnector	:= fbMachineControl
									);
	fbPrepareScreen					: FB_MCHMIPrepareDataForScreen;
	fbPrepareScreen_00_01			: FB_MCHMIPrepareDataForScreen_00_01;
	fbPrepareScreen_00_02			: FB_MCHMIPrepareDataForScreen_00_02;
	fbPrepareScreen_00_03			: FB_MCHMIPrepareDataForScreen_00_03;
	fbPrepareScreen_00_04			: FB_MCHMIPrepareDataForScreen_00_04;
	fbPrepareScreen_00_05			: FB_MCHMIPrepareDataForScreen_00_05;
	
	fbPrepareScreen_01_XX			: FB_MCHMIPrepareDataForScreen_01_XX;
	fbPrepareScreen_02_XX			: FB_MCHMIPrepareDataForScreen_02_XX;
	fbPrepareScreen_03_XX			: FB_MCHMIPrepareDataForScreen_03_XX;
	fbPrepareScreen_04_XX			: FB_MCHMIPrepareDataForScreen_04_XX;
	fbPrepareScreen_05_XX			: FB_MCHMIPrepareDataForScreen_05_XX;
	fbPrepareScreen_06_XX			: FB_MCHMIPrepareDataForScreen_06_XX;
	fbPrepareScreen_07_XX			: FB_MCHMIPrepareDataForScreen_07_XX;
	
END_VAR

END_PROGRAM

// ---- POUs/01_MC/FB_MCHMIMachineControl_HMI.TcPOU
(*			
	RafalOS
	Rafał Osajda		20.11.2025		TC 4024.66
	Łącznik MachineControl do wizualizacji
*)
FUNCTION_BLOCK FB_MCHMIMachineControl_HMI EXTENDS FB_BaseTopElement_HMI IMPLEMENTS ITF_MCHMIMachineControl_HMI, ITF_MCHMIMachineControl_HMI_PrepScr					
VAR
	(*	Główny łacznik do logiki maszyny	*)
	itfMachineControlConnector			: ITF_MCMachineControl_HMI_Connector;
	refstMachineControlData				: REFERENCE TO ST_MCHMIMachineControl_HMI;
	(*	Moduł Receptur	*)
	itfRecipe							: ITF_BaseRecipe_HMI;
	(*	Przygotowywanie danych dla ramek	*)
	arrPrepareScreen					: ARRAY [1..20] OF ITF_MCHMIPrepareScreen_Init;
	iNumberOfAddedPrepScren				: INT;
	arrPrepareScreen_Execute			: ARRAY [0..GVL_HMIEConstans.MAX_NUMBER_OF_BUTTON_IN_MENU] OF 
											ARRAY [0..GVL_SaMConstans.NUMBER_OF_MODES] OF ITF_MCHMIPrepareDataForScreen;
	refstHMICommonData					: REFERENCE TO ST_MCHMICommonData;
	(*	wspólne opisy *)
	stRecipeInfoSelect			: ST_BaseLabel;
	stRecipeInfoNotSelect		: ST_BaseLabel;
	
END_VAR

METHOD PUBLIC AddPrepareScreenModuleFromManager : BOOL
VAR_INPUT
	itfModule	: ITF_MCHMIPrepareScreen_Init;// ITF_MCHMIPrepareDataForScreen;
END_VAR
IF (THIS^.iNumberOfAddedPrepScren + 1 <= 20) THEN
	THIS^.AddComponent (itfComponentHMI := itfModule);
	THIS^.iNumberOfAddedPrepScren := THIS^.iNumberOfAddedPrepScren + 1;
	THIS^.arrPrepareScreen [THIS^.iNumberOfAddedPrepScren] := itfModule;
	AddPrepareScreenModuleFromManager := TRUE;
ELSE
	AddPrepareScreenModuleFromManager := FALSE;
END_IF
END_METHOD

(*			
	RafalOS
	Rafał Osajda		03.03.2025		TC 4026.13		wer. 0.0.0.1
	Kopiuje składniki z wybranej receptury i tworzy nową recepture
*)
METHOD PUBLIC AddRecipeFromRecipe : BOOL
VAR_INPUT
	uiNumberRecipe				: UINT;
	stTexts						: ST_BaseLabel;
END_VAR
THIS^.itfRecipe.AddRecipeFromRecipe (
	uiNumberRecipe		:= uiNumberRecipe,
	stTexts				:= stTexts
);
END_METHOD

(*			
	RafalOS
	Rafał Osajda		03.03.2025		TC 4026.13		wer. 0.0.0.1
	Kopiuje składniki z wybranego szablonu i tworzy nową recepture
*)
METHOD PUBLIC AddRecipeFromTemplate : BOOL
VAR_INPUT
	uiNumberTemplates			: UINT;
	stTexts						: ST_BaseLabel;
END_VAR
THIS^.itfRecipe.AddRecipeFromTemplate (
	uiNumberTemplates	:= uiNumberTemplates,
	stTexts				:= stTexts
);
END_METHOD

(*			
	RafalOS
	Rafał Osajda		26.11.2025		TC 4024.66
	Podłaczenie modułu receptur
*)
METHOD PUBLIC AddRecipeModulFormManager : BOOL
VAR_INPUT
	fbRecipeModul		: ITF_BaseRecipe_HMI;
END_VAR
THIS^.itfRecipe := fbRecipeModul;
END_METHOD

(*			
	RafalOS
	Rafał Osajda		19.11.2025		TC 4024.66
	Sprzątanie po stronie wywoływane z HMIManager i wywołująca odpowiednią metode z ITF z arrPrepareScreen
*)
METHOD ClearAfterScreenFroHMIManager : BOOL
VAR_INPUT
	iScreen		: INT;
	iMode		: INT;
END_VAR
IF (THIS^.arrPrepareScreen_Execute [iScreen][iMode] <> 0) THEN
	THIS^.arrPrepareScreen_Execute [iScreen][iMode].ClearAfterScreen ();
END_IF
END_METHOD

(*			
	RafalOS
	Rafał Osajda		03.06.2025		TC 4024.66
	usuwa referencje do wybranej
*)
METHOD PUBLIC ClearChosen
VAR_INPUT
END_VAR
THIS^.itfRecipe.ClearChosen ();
END_METHOD

(*			
	RafalOS
	Rafał Osajda		25.10.2025		TC 4024.66
	Utworzenie nowych szablonów receptur na podstawie dodanych fb zewnętrznych - wywołanie metody powoduje
	skosowanie dotychczasowych szablonów i receptur
*)
METHOD PUBLIC CreateRecipeTemplates : BOOL
VAR_INPUT
END_VAR
THIS^.itfRecipe.CreateRecipeTemplates ();
END_METHOD

(*			
	RafalOS
	Rafał Osajda		03.03.2025		TC 4026.13		wer. 0.0.0.1
	
*)
METHOD PUBLIC DeleteRecipe : BOOL
VAR_INPUT
	uiNumber				: uint;
END_VAR
THIS^.itfRecipe.DeleteRecipe (uiNumber := uiNumber);
END_METHOD

METHOD FB_init : BOOL
VAR_INPUT
	bInitRetains : BOOL; // if TRUE, the retain variables are initialized (warm start / cold start)
	bInCopyCode : BOOL;  // if TRUE, the instance afterwards gets moved into the copy code (online change)
	itfBaseLoggerConnector				: ITF_BaseLogger_HMI_Connector;	//bezpośredni łącznik do logera
	itfMachineControlConnector			: ITF_MCMachineControl_HMI_Connector;
END_VAR
//Przypisanie do elementu który własnie stworzyliśmy
THIS^.itfMachineControlConnector := itfMachineControlConnector;
//Przypisanie do elementów z biblioteki
THIS^.itfBaseLoggerElementConnector := itfMachineControlConnector;
THIS^.itfBaseComponentConnector := itfMachineControlConnector;
THIS^.itfBaseControlElementConnector := itfMachineControlConnector;
THIS^.itfBaseGroupElementConnector := itfMachineControlConnector;
THIS^.itfBaseTopElementConnector := itfMachineControlConnector;
//
THIS^.itfBaseLoggerConnector := itfBaseLoggerConnector;

IF (THIS^.itfMachineControlConnector <> 0 AND
	THIS^.itfBaseLoggerElementConnector <> 0 AND
	THIS^.itfBaseComponentConnector	<> 0 AND
	THIS^.itfBaseControlElementConnector <> 0 AND
	THIS^.itfBaseGroupElementConnector <> 0 AND
	THIS^.itfBaseTopElementConnector <> 0 AND
	THIS^.itfBaseLoggerConnector <> 0) THEN
	THIS^.bIsInit						:= TRUE;
END_IF

THIS^.SetText (eLocation := E_BaseLocation.pl, wsDescription := "Receptura wybrana");
THIS^.SetText (eLocation := E_BaseLocation.en, wsDescription := "Recipe selected");
THIS^.SetText (eLocation := E_BaseLocation.de, wsDescription := "Rezept ausgewählt");
THIS^.stRecipeInfoSelect := THIS^.GetTexts ();

THIS^.SetText (eLocation := E_BaseLocation.pl, wsDescription := "Brak wybranej receptury");
THIS^.SetText (eLocation := E_BaseLocation.en, wsDescription := "No recipe selected");
THIS^.SetText (eLocation := E_BaseLocation.de, wsDescription := "Kein Rezept ausgewählt");
THIS^.stRecipeInfoNotSelect := THIS^.GetTexts ();
END_METHOD

METHOD GetActiveMode : E_BaseMachineMode
VAR_INPUT
END_VAR
GetActiveMode := THIS^.itfMachineControlConnector.GetActiveMode ();
END_METHOD

METHOD PUBLIC GetActiveModeFromManager : E_BaseMachineMode
VAR_INPUT
END_VAR
GetActiveModeFromManager := THIS^.itfMachineControlConnector.GetActiveMode ();
END_METHOD

METHOD PUBLIC GetActiveModeName : ST_BaseLabel
VAR_INPUT
END_VAR
GetActiveModeName := THIS^.itfMachineControlConnector.GetActiveModeName ();
END_METHOD

METHOD GetActiveState : E_BaseMachineState
VAR_INPUT
END_VAR
GetActiveState := THIS^.itfMachineControlConnector.GetActiveState ();
END_METHOD

METHOD PUBLIC GetActiveStateName : ST_BaseLabel
VAR_INPUT
END_VAR
GetActiveStateName := THIS^.itfMachineControlConnector.GetActiveStateName ();
END_METHOD

(*			
	RafalOS
	Rafał Osajda		17.12.2025		TC 4024.66
	Pobiera listę elementów które posiadaja parametr i 
	przypisuje ja do zadanej struktury i zwraca true jak się uda
*)
METHOD GetElementNamesWithParameter : BOOL
VAR_INPUT
	stDane			: REFERENCE TO ST_MCElementListWithParameter;
END_VAR
GetElementNamesWithParameter := THIS^.itfMachineControlConnector.GetElementNamesWithParameter (
									stDane := stDane
								);
END_METHOD

(*			
	RafalOS
	Rafał Osajda		07.12.2025		TC 4024.66
	Pobierz informacje o aktualnym stanie recepur tzn o tym czy jest wybrana a jak tak to która
*)
METHOD PUBLIC GetInformationLatestRecipes
VAR_INST
	tonChangeSelectRecipe	: TON;
	rtNewRecipeSelected		: R_TRIG;
	ftNewRecipeSelected		: F_TRIG;
END_VAR
THIS^.refstHMICommonData.stRecipeInformation.bRecipeSelected := THIS^.itfRecipe.IsRecipeSelected ();
rtNewRecipeSelected (CLK := THIS^.refstHMICommonData.stRecipeInformation.bRecipeSelected);
ftNewRecipeSelected (CLK := THIS^.refstHMICommonData.stRecipeInformation.bRecipeSelected);
tonChangeSelectRecipe (PT := T#3S);

IF (rtNewRecipeSelected.Q OR 
	THIS^.refstHMICommonData.stRecipeInformation.bNewSelectedRecipe) THEN
	;//jest wybrana
	THIS^.refstHMICommonData.stRecipeInformation.bNewSelectedRecipe := FALSE;
	tonChangeSelectRecipe.IN := TRUE;
	THIS^.refstHMICommonData.stRecipeInformation.dwBackgroud := 16#FF00FF00;//zielony
	THIS^.refstHMICommonData.stRecipeInformation.dwText := 16#FF000000;//cxzarny
	THIS^.refstHMICommonData.stRecipeInformation.wsRecipeInformation := THIS^.GetTextFromLabelForActiveLocation (stLabel := THIS^.stRecipeInfoSelect);
END_IF
IF (ftNewRecipeSelected.Q) THEN
	THIS^.refstHMICommonData.stRecipeInformation.dwBackgroud := 16#FFFF0000; //czerwony
	THIS^.refstHMICommonData.stRecipeInformation.dwText := 16#FFFFFF00;//zółty
	THIS^.refstHMICommonData.stRecipeInformation.wsRecipeInformation := THIS^.GetTextFromLabelForActiveLocation (stLabel := THIS^.stRecipeInfoNotSelect);
END_IF
IF (tonChangeSelectRecipe.Q) THEN 
	tonChangeSelectRecipe.IN := FALSE;
	THIS^.refstHMICommonData.stRecipeInformation.bNewSelectedRecipe := FALSE;
	THIS^.refstHMICommonData.stRecipeInformation.dwBackgroud := 16#FF00FF00;//zielony
	THIS^.refstHMICommonData.stRecipeInformation.dwText := 16#FF000000;//cxzarny
	THIS^.refstHMICommonData.stRecipeInformation.wsRecipeInformation := THIS^.GetNumberAndNameRecipe ();
END_IF
END_METHOD

(*			
	RafalOS
	Rafał Osajda		03.03.2025		TC 4026.13		wer. 0.0.0.1
	
*)
METHOD PUBLIC GetIngredientFromRecipe : ST_BaseDescriptor
VAR_INPUT
	uiNumberOfRecipe			: UINT;
	uiNumberOfIngredient		: UINT;
END_VAR
GetIngredientFromRecipe			:= THIS^.itfRecipe.GetIngredientFromRecipe (
									uiNumberOfRecipe := uiNumberOfRecipe,
									uiNumberOfIngredient := uiNumberOfIngredient
								);
END_METHOD

(*			
	RafalOS
	Rafał Osajda		02.12.2025		TC 4024.66
	Zwraca do tablicy wybrany zakres składników
*)
METHOD PUBLIC GetIngredientRange 
VAR_INPUT
	iRecipe			: INT;	//numer receptury z której bierzemy składniki
	iStartIndex		: INT;	//numer startowy składnika
	iCount			: INT;	//ilośc pobieranych 
END_VAR
VAR_IN_OUT
	arrOut : ARRAY [*] OF ST_BaseDescriptor;
END_VAR
VAR_OUTPUT
	iNumberOfFilledData	: INT;	//ilosc wypelnionych danych na strone
END_VAR
THIS^.itfRecipe.GetIngredientRange (
	iRecipe		:= iRecipe,
	iStartIndex	:= iStartIndex,
	iCount		:= iCount,
	arrOut		:= arrOut,
	iNumberOfFilledData => iNumberOfFilledData
);
END_METHOD

METHOD PUBLIC GetListOfNameRecipe : ST_BaseRecipeList
VAR_INPUT
END_VAR
GetListOfNameRecipe := THIS^.itfRecipe.GetNameList ();
END_METHOD

METHOD PUBLIC GetListOfNameTemplate : ST_BaseRecipeList
VAR_INPUT
END_VAR
GetListOfNameTemplate := THIS^.itfRecipe.GetNameListTemplate ();
END_METHOD

(*			
	RafalOS
	Rafał Osajda		25.11.2025		TC 4024.66
	Zwraca nazwę trybu o zadanym numerze
*)
METHOD GetModeName : ST_BaseLabel
VAR_INPUT
	iMode	: INT;
END_VAR
GetModeName := THIS^.itfMachineControlConnector.GetModeName (iNumber := iMode);
END_METHOD

(*			
	RafalOS
	Rafał Osajda		07.12.2025		TC 4024.66
	Pobiera nazwę i numer aktualnej receptury
*)
METHOD PRIVATE GetNumberAndNameRecipe : WSTRING
VAR_INPUT
END_VAR

VAR
	wsNumber	: WSTRING;
	wsName		: WSTRING;
	wsResult	: WSTRING;
END_VAR
wsNumber := TO_WSTRING (THIS^.itfRecipe.GetNumberOfChoosen ());
wsName := THIS^.GetTextFromLabelForActiveLocation (stLabel := THIS^.itfRecipe.GetNamesOfSelectRecipe ());

wsResult := wconcat (WCONCAT (" ID - ", wsNumber), WCONCAT (" - " ,wsName));


GetNumberAndNameRecipe := wsResult;
END_METHOD

(*			
	RafalOS
	Rafał Osajda		03.03.2025		TC 4026.13		wer. 0.0.0.1
	
*)
METHOD PUBLIC GetNumberIngredientOfRecipe : UINT
VAR_INPUT
	uiNumber				: UINT;
END_VAR
GetNumberIngredientOfRecipe 		:= THIS^.itfRecipe.GetNumberIngredientOfRecipe (uiNumber := uiNumber);
END_METHOD

METHOD PUBLIC GetNumberOfChoosen : UINT
VAR_INPUT
END_VAR
GetNumberOfChoosen := THIS^.itfRecipe.GetNumberOfChoosen ();
END_METHOD

METHOD PUBLIC GetNumberOfRecipe : UINT
VAR_INPUT
END_VAR
GetNumberOfRecipe			:= THIS^.itfRecipe.GetNumberOfRecipe ();
END_METHOD

METHOD PUBLIC GetNumberOfTemplate : UINT
VAR_INPUT
END_VAR
GetNumberOfTemplate		:= THIS^.itfRecipe.GetNumberOfTemplate ();
END_METHOD

METHOD GetStateName : ST_BaseLabel
VAR_INPUT
	iNumber		: INT;
END_VAR
GetStateName := THIS^.itfMachineControlConnector.GetStateName (iNumber := iNumber);
END_METHOD

METHOD GetStateTimeForMode : LTIME
VAR_INPUT
	iMode		: INT;
	iState		: INT;
END_VAR
GetStateTimeForMode := THIS^.itfMachineControlConnector.GetStateTimeForMode (iMode := iMode, iState := iState);
END_METHOD

METHOD GetTimeWorkForMode : LTIME
VAR_INPUT
	iMode	: INT;
END_VAR
GetTimeWorkForMode := THIS^.itfMachineControlConnector.GetTimeWorkForMode (iMode := iMode);
END_METHOD

(*			
	RafalOS
	Rafał Osajda		25.11.2025		TC 4024.66
	Zwraca całkowity czas pracy maszyny
*)
METHOD PUBLIC GetTotalWorkTime : LTIME
VAR_INPUT
END_VAR
GetTotalWorkTime := THIS^.itfMachineControlConnector.GetTotalWorkTime ();
END_METHOD

(*			
	RafalOS
	Rafał Osajda		25.11.2025		TC 4024.66
	Zwraca czy zmiana stanu się skońćzyła
*)
METHOD IsChangeModeDone : BOOL
VAR_INPUT
END_VAR
IsChangeModeDone := this^.itfMachineControlConnector.IsChangeModeDone ();
END_METHOD

(*			
	RafalOS
	Rafał Osajda		25.11.2025		TC 4024.66
	Zwraca czy tryb o podanym numerze jest włączony
*)
METHOD IsModeEnabled : BOOL
VAR_INPUT
	iMode 	: INT;
END_VAR
IsModeEnabled := THIS^.itfMachineControlConnector.IsModeEnabled (iMode := iMode);
END_METHOD

METHOD IsStateActive : BOOL
VAR_INPUT
	iTestState : INT;
END_VAR
IsStateActive := THIS^.itfMachineControlConnector.IsStateIsActual (iTestState := iTestState);
END_METHOD

METHOD IsStateEnableInMode : BOOL
VAR_INPUT
	iTestState	: INT;
END_VAR
IsStateEnableInMode := THIS^.itfMachineControlConnector.IsStateActiveInCurrentMode ();
END_METHOD

METHOD PUBLIC LinkMachineControlData : BOOL
VAR_INPUT
	stData			: REFERENCE TO ST_MCHMIMachineControl_HMI_Link;
END_VAR
THIS^.refstMachineControlData REF= stData.stMachineControl;

//w tablicy pole 1 zajmuje metoda pusta domyślna do niej się nie linkuje danych
THIS^.arrPrepareScreen [2].LinkDataHMI_00_01 (refstData := stData.stPrepScr_00_01);
THIS^.arrPrepareScreen [3].LinkDataHMI_00_02 (refstData := stData.stPrepScr_00_02);
THIS^.arrPrepareScreen [4].LinkDataHMI_00_03 (refstData := stData.stPrepScr_00_03);
THIS^.arrPrepareScreen [5].LinkDataHMI_00_04 (refstData := stData.stPrepScr_00_04);
THIS^.arrPrepareScreen [6].LinkDataHMI_00_05 (refstData := stData.stPrepScr_00_05);

THIS^.arrPrepareScreen [7].LinkDataHMI_01_XX (refstData := stData.stPrepScr_01_XX);
THIS^.arrPrepareScreen [8].LinkDataHMI_02_XX (refstData := stData.stPrepScr_02_XX);
THIS^.arrPrepareScreen [9].LinkDataHMI_03_XX (refstData := stData.stPrepScr_03_XX);
THIS^.arrPrepareScreen [10].LinkDataHMI_04_XX (refstData := stData.stPrepScr_04_XX);
THIS^.arrPrepareScreen [11].LinkDataHMI_05_XX (refstData := stData.stPrepScr_05_XX);
THIS^.arrPrepareScreen [12].LinkDataHMI_06_XX (refstData := stData.stPrepScr_06_XX);
THIS^.arrPrepareScreen [13].LinkDataHMI_07_XX (refstData := stData.stPrepScr_07_XX);

THIS^.refstHMICommonData REF= stData.stCommonData;
THIS^.arrPrepareScreen [2].LinkHMICommonData (stHMICommonData := stData.stCommonData);
THIS^.arrPrepareScreen [3].LinkHMICommonData (stHMICommonData := stData.stCommonData);
THIS^.arrPrepareScreen [4].LinkHMICommonData (stHMICommonData := stData.stCommonData);
THIS^.arrPrepareScreen [5].LinkHMICommonData (stHMICommonData := stData.stCommonData);
THIS^.arrPrepareScreen [6].LinkHMICommonData (stHMICommonData := stData.stCommonData);
THIS^.arrPrepareScreen [7].LinkHMICommonData (stHMICommonData := stData.stCommonData);
THIS^.arrPrepareScreen [8].LinkHMICommonData (stHMICommonData := stData.stCommonData);
THIS^.arrPrepareScreen [9].LinkHMICommonData (stHMICommonData := stData.stCommonData);
THIS^.arrPrepareScreen [10].LinkHMICommonData (stHMICommonData := stData.stCommonData);
THIS^.arrPrepareScreen [11].LinkHMICommonData (stHMICommonData := stData.stCommonData);
THIS^.arrPrepareScreen [12].LinkHMICommonData (stHMICommonData := stData.stCommonData);
THIS^.arrPrepareScreen [13].LinkHMICommonData (stHMICommonData := stData.stCommonData);

THIS^.itfRecipe.LinkRecipeDataHMI (stRecipe := stData.stRecipe);

THIS^.refstBaseLoggerElementDataHMI REF= stData.stBaseLoggerElement;
THIS^.refstBaseComponentDataHMI REF= stData.stBaseComponent;
THIS^.refstBaseControlElementDataHMI REF= stData.stBaseControlElement;
THIS^.refstBaseGroupElementDataHMI REF= stData.stBaseGroupElement;
THIS^.refstBaseTopElementDataHMI REF= stData.stBaseTopElement;


THIS^.CreateLinkToEventsMemory ();

IF (__ISVALIDREF (THIS^.refstMachineControlData) AND THIS^.IsLinkedReferences ()) THEN
	THIS^.bIsValidData := TRUE;
	LinkMachineControlData := TRUE;
END_IF
END_METHOD

(*			
	RafalOS
	Rafał Osajda		20.11.2025		TC 4024.66
	Podpięcie modułu generowania danych do odpowiedniej pozycji w tablicy [Okno][Tryb]
*)
METHOD PUBLIC LinkPrepareScreenToArrayFromConfiguration : BOOL
VAR_INPUT
	iScreen		: INT;
	iMode		: INT;
	itfModule	: ITF_MCHMIPrepareDataForScreen;
END_VAR
THIS^.arrPrepareScreen_Execute [iScreen][iMode] := itfModule;
END_METHOD

(*			
	RafalOS
	Rafał Osajda		14.11.2025		TC 4024.66
	Metoda przygotowywania danych dla HMI 
	W niej odbywa się odpytywanie właściego elementu przez łącznik
*)
METHOD PUBLIC PrepareDataForHMI : BOOL
VAR
	iJ		: INT;
END_VAR



SUPER^.PrepareDataForHMI ();
END_METHOD

(*			
	RafalOS
	Rafał Osajda		19.11.2025		TC 4024.66
	Przygotowanie danych dla strony wywoływane z HMIManager i wywołująca odpowiednią metode z ITF z arrPrepareScreen
*)
METHOD PrepareDataForScreenFromHMIManager : BOOL
VAR_INPUT
	iScreen		: INT;
	iMode		: INT;
END_VAR
THIS^.refstHMICommonData.wsActualMode := THIS^.GetTextFromLabelForActiveLocation (THIS^.itfMachineControlConnector.GetActiveModeName ());
THIS^.refstHMICommonData.wsActualState := THIS^.GetTextFromLabelForActiveLocation (THIS^.itfMachineControlConnector.GetActiveStateName ());

IF (THIS^.arrPrepareScreen_Execute [iScreen][iMode] <> 0) THEN
	THIS^.arrPrepareScreen_Execute [iScreen][iMode].PrepareDataForHMI ();
END_IF
END_METHOD

(*			
	RafalOS
	Rafał Osajda		19.11.2025		TC 4024.66
	Przygotowanie strony wywoływane z HMIManager i wywołująca odpowiednią metode z ITF z arrPrepareScreen
*)
METHOD PrepareForScreenFromHMIManager : BOOL
VAR_INPUT
	iScreen		: INT;
	iMode		: INT;
END_VAR
IF (THIS^.arrPrepareScreen_Execute [iScreen][iMode] <> 0) THEN
	THIS^.arrPrepareScreen_Execute [iScreen][iMode].PrepareForScreen ();
END_IF
END_METHOD

(*			
	RafalOS
	Rafał Osajda		06.12.2025		TC 4024.66
	Wybranie receputury
*)
METHOD SelectRecipe : BOOL
VAR_INPUT
	uiRecipe: UINT;
END_VAR
THIS^.itfRecipe.SelectRecipe (
	uiRecipe := uiRecipe
);
END_METHOD

(*			
	RafalOS
	Rafał Osajda		20.11.2025		TC 4024.66
	Ustawienei zmiennej w wspólnych zmiennych z managera
*)
METHOD PUBLIC SetChangePageFromManager : BOOL
VAR_INPUT
	bValue	: BOOL;
END_VAR
THIS^.refstHMICommonData.bChangePage := bValue;
END_METHOD

(*			
	RafalOS
	Rafał Osajda		24.11.2025		TC 4024.66
	Zmien tryb
*)
METHOD SetCmdChangeMode : BOOL
VAR_INPUT
	eCmdNumber	: E_SaMCommandChangeMode;
END_VAR
THIS^.itfMachineControlConnector.SetCmdChangeMode (eCmdNumber := eCmdNumber);
END_METHOD

(*			
	RafalOS
	Rafał Osajda		24.11.2025		TC 4024.66
	Zmien stan 
*)
METHOD public SetCmdChangeState : BOOL
VAR_INPUT
	eCmdNumber : E_SaMCommandChangeState;
END_VAR
THIS^.itfMachineControlConnector.SetCmdChangeState (eCmdNumber := eCmdNumber);
END_METHOD

(*			
	RafalOS
	Rafał Osajda		05.12.2025		TC 4024.66
	Ustawia nową wartośc w podanym składniku
*)
METHOD PUBLIC SetIngredientValue
VAR_INPUT
	iRecipe			: int;
	iIngredient		: INT;
	rValue			: REAL;
END_VAR
THIS^.itfRecipe.SetIngredientValue (
	iRecipe := iRecipe,
	iIngredient := iIngredient,
	rValue := rValue
);
END_METHOD

END_FUNCTION_BLOCK

// ---- POUs/02_PrepareScreenParent/FB_MCHMIPrepareDataForScreen.TcPOU
(*			
	RafalOS
	Rafał Osajda		19.11.2025		TC 4024.66
	Domyślne przygotowanie danych dla ekranu
*)
FUNCTION_BLOCK FB_MCHMIPrepareDataForScreen EXTENDS FB_BaseComponent_HMI IMPLEMENTS ITF_MCHMIPrepareScreen_Init
VAR
	//itf do lacznika machinecontrol
	//strulture danych 
	itfExtendedDisplay			: ITF_MCHMIDisplayExtension;
	refstHMICommonData			: reference to ST_MCHMICommonData;
END_VAR

(*			
	RafalOS
	Rafał Osajda		19.11.2025		TC 4024.66
	Czyści danych przy zmienia ramki po poprzedniej ramce
*)
METHOD PUBLIC ClearAfterScreen : BOOL
VAR_INPUT
END_VAR
IF (THIS^.itfExtendedDisplay <> 0) THEN
	THIS^.itfExtendedDisplay.ExtendedClearAfterScreen ();
END_IF
END_METHOD

METHOD PUBLIC LinkDataHMI_00_01 : BOOL
VAR_INPUT
	refstData				: REFERENCE TO ST_MCHMIPrepareScreen_00_01;
END_VAR
END_METHOD

METHOD PUBLIC LinkDataHMI_00_02 : BOOL
VAR_INPUT
	refstData				: REFERENCE TO ST_MCHMIPrepareScreen_00_02;
END_VAR
END_METHOD

METHOD PUBLIC LinkDataHMI_00_03 : BOOL
VAR_INPUT
	refstData				: REFERENCE TO ST_MCHMIPrepareScreen_00_03;
END_VAR
END_METHOD

METHOD PUBLIC LinkDataHMI_00_04 : BOOL
VAR_INPUT
	refstData				: REFERENCE TO ST_MCHMIPrepareScreen_00_04;
END_VAR
END_METHOD

METHOD PUBLIC LinkDataHMI_00_05 : BOOL
VAR_INPUT
	refstData				: REFERENCE TO ST_MCHMIPrepareScreen_00_05;
END_VAR
END_METHOD

METHOD PUBLIC LinkDataHMI_01_XX : BOOL
VAR_INPUT
	refstData				: REFERENCE TO ST_MCHMIPrepareScreen_01_XX;
END_VAR
END_METHOD

METHOD PUBLIC LinkDataHMI_02_XX : BOOL
VAR_INPUT
	refstData				: REFERENCE TO ST_MCHMIPrepareScreen_02_XX;
END_VAR
END_METHOD

METHOD PUBLIC LinkDataHMI_03_XX : BOOL
VAR_INPUT
	refstData				: REFERENCE TO ST_MCHMIPrepareScreen_03_XX;
END_VAR
END_METHOD

METHOD PUBLIC LinkDataHMI_04_XX : BOOL
VAR_INPUT
	refstData				: REFERENCE TO ST_MCHMIPrepareScreen_04_XX;
END_VAR
END_METHOD

METHOD PUBLIC LinkDataHMI_05_XX : BOOL
VAR_INPUT
	refstData				: REFERENCE TO ST_MCHMIPrepareScreen_05_XX;
END_VAR
END_METHOD

METHOD PUBLIC LinkDataHMI_06_XX : BOOL
VAR_INPUT
	refstData				: REFERENCE TO ST_MCHMIPrepareScreen_06_XX;
END_VAR
END_METHOD

METHOD PUBLIC LinkDataHMI_07_XX : BOOL
VAR_INPUT
	refstData				: REFERENCE TO ST_MCHMIPrepareScreen_07_XX;
END_VAR
END_METHOD

METHOD PUBLIC LinkExtensionDisplay : BOOL
VAR_INPUT
	fbExtendedDisplay			: ITF_MCHMIDisplayExtension;
END_VAR
THIS^.itfExtendedDisplay := fbExtendedDisplay;
END_METHOD

(*			
	RafalOS
	Rafał Osajda		20.11.2025		TC 4024.66
	Podłączenie wspólnych danych do modułu 
*)
METHOD PUBLIC LinkHMICommonData : BOOL
VAR_INPUT
	stHMICommonData	: REFERENCE TO ST_MCHMICommonData;
END_VAR
this^.refstHMICommonData ref= stHMICommonData;
END_METHOD

(*			
	RafalOS
	Rafał Osajda		14.11.2025		TC 4024.66
	Metoda przygotowywania danych dla HMI 
	W niej odbywa się odpytywanie właściego elementu przez łącznik
*)
METHOD PUBLIC PrepareDataForHMI : BOOL
VAR_INPUT
END_VAR
IF (THIS^.itfExtendedDisplay <> 0) THEN
	THIS^.itfExtendedDisplay.ExtendedPrepareDataForHMI ();
END_IF
END_METHOD

(*			
	RafalOS
	Rafał Osajda		19.11.2025		TC 4024.66
	Przygotowanie ramki pood tamke do wyświetlenia - tylko przygotowanie a nie przygotowanie danych do wyświetlenia
*)
METHOD PUBLIC PrepareForScreen : BOOL
VAR_INPUT
END_VAR
IF (THIS^.itfExtendedDisplay <> 0) THEN
	THIS^.itfExtendedDisplay.ExtendedPrepareForScreen ();
END_IF
END_METHOD

END_FUNCTION_BLOCK

// ---- POUs/03_MW_Production/FB_MCHMIPrepareDataForScreen_00_01.TcPOU
(*			
	RafalOS
	Rafał Osajda		20.11.2025		TC 4024.66
	Moduł przygotowania danych dla Okna głównego w trybie produkcji
*)
FUNCTION_BLOCK FB_MCHMIPrepareDataForScreen_00_01 EXTENDS FB_MCHMIPrepareDataForScreen IMPLEMENTS ITF_MCHMIPrepareDataForScreen
VAR
	itfMachineControlHMI	: ITF_MCHMIMachineControl_HMI_PrepScr_00_01;
	refstData				: REFERENCE TO ST_MCHMIPrepareScreen_00_01;
END_VAR

(*			
	RafalOS
	Rafał Osajda		19.11.2025		TC 4024.66
	Czyści danych przy zmienia ramki po poprzedniej ramce
*)
METHOD PUBLIC ClearAfterScreen : BOOL
VAR_INPUT
END_VAR
SUPER^.ClearAfterScreen ();
END_METHOD

METHOD PUBLIC LinkDataHMI_00_01 : BOOL
VAR_INPUT
	refstData				: REFERENCE TO ST_MCHMIPrepareScreen_00_01;
END_VAR
THIS^.refstData REF= refstData;
END_METHOD

METHOD PUBLIC LinkMachineControlHMI : BOOL
VAR_INPUT
	fbMachineControlHMI	: ITF_MCHMIMachineControl_HMI_PrepScr_00_01;
END_VAR
this^.itfMachineControlHMI := fbMachineControlHMI;
END_METHOD

(*			
	RafalOS
	Rafał Osajda		14.11.2025		TC 4024.66
	Metoda przygotowywania danych dla HMI 
	W niej odbywa się odpytywanie właściego elementu przez łącznik
*)
METHOD PUBLIC PrepareDataForHMI : BOOL
VAR_INPUT
END_VAR
SUPER^.PrepareDataForHMI ();
END_METHOD

(*			
	RafalOS
	Rafał Osajda		19.11.2025		TC 4024.66
	Przygotowanie ramki pood tamke do wyświetlenia - tylko przygotowanie a nie przygotowanie danych do wyświetlenia
*)
METHOD PUBLIC PrepareForScreen : BOOL
VAR_INPUT
END_VAR
SUPER^.PrepareForScreen ();
END_METHOD

END_FUNCTION_BLOCK

// ---- POUs/04_MW_Maitenance/FB_MCHMIPrepareDataForScreen_00_02.TcPOU
(*			
	RafalOS
	Rafał Osajda		20.11.2025		TC 4024.66
	Moduł przygotowania danych dla Okna głównego w trybie konserwacji
*)
FUNCTION_BLOCK FB_MCHMIPrepareDataForScreen_00_02 EXTENDS FB_MCHMIPrepareDataForScreen IMPLEMENTS ITF_MCHMIPrepareDataForScreen
VAR
	itfMachineControlHMI	: ITF_MCHMIMachineControl_HMI_PrepScr_00_02;
	refstData				: REFERENCE TO ST_MCHMIPrepareScreen_00_02;
	
END_VAR

(*			
	RafalOS
	Rafał Osajda		19.11.2025		TC 4024.66
	Czyści danych przy zmienia ramki po poprzedniej ramce
*)
METHOD PUBLIC ClearAfterScreen : BOOL
VAR_INPUT
END_VAR
SUPER^.ClearAfterScreen ();
END_METHOD

METHOD PUBLIC LinkDataHMI_00_02 : BOOL
VAR_INPUT
	refstData				: REFERENCE TO ST_MCHMIPrepareScreen_00_02;
END_VAR
THIS^.refstData REF= refstData;
END_METHOD

METHOD PUBLIC LinkMachineControlHMI : BOOL
VAR_INPUT
	fbMachineControlHMI	: ITF_MCHMIMachineControl_HMI_PrepScr_00_02;
END_VAR
this^.itfMachineControlHMI := fbMachineControlHMI;
END_METHOD

(*			
	RafalOS
	Rafał Osajda		14.11.2025		TC 4024.66
	Metoda przygotowywania danych dla HMI 
	W niej odbywa się odpytywanie właściego elementu przez łącznik
*)
METHOD PUBLIC PrepareDataForHMI : BOOL
VAR_INPUT
END_VAR
SUPER^.PrepareDataForHMI ();
END_METHOD

(*			
	RafalOS
	Rafał Osajda		19.11.2025		TC 4024.66
	Przygotowanie ramki pood tamke do wyświetlenia - tylko przygotowanie a nie przygotowanie danych do wyświetlenia
*)
METHOD PUBLIC PrepareForScreen : BOOL
VAR_INPUT
END_VAR
SUPER^.PrepareForScreen ();
END_METHOD

END_FUNCTION_BLOCK

// ---- POUs/05_MW_Manual/FB_MCHMIPrepareDataForScreen_00_03.TcPOU
(*			
	RafalOS
	Rafał Osajda		20.11.2025		TC 4024.66
	Moduł przygotowania danych dla Okna głównego w trybie ręcznym
*)
FUNCTION_BLOCK FB_MCHMIPrepareDataForScreen_00_03 EXTENDS FB_MCHMIPrepareDataForScreen IMPLEMENTS ITF_MCHMIPrepareDataForScreen
VAR
	itfMachineControlHMI	: ITF_MCHMIMachineControl_HMI_PrepScr_00_03;
	refstData				: REFERENCE TO ST_MCHMIPrepareScreen_00_03;
END_VAR

(*			
	RafalOS
	Rafał Osajda		19.11.2025		TC 4024.66
	Czyści danych przy zmienia ramki po poprzedniej ramce
*)
METHOD PUBLIC ClearAfterScreen : BOOL
VAR_INPUT
END_VAR
SUPER^.ClearAfterScreen ();
END_METHOD

METHOD PUBLIC LinkDataHMI_00_03 : BOOL
VAR_INPUT
	refstData				: REFERENCE TO ST_MCHMIPrepareScreen_00_03;
END_VAR
THIS^.refstData REF= refstData;
END_METHOD

METHOD PUBLIC LinkMachineControlHMI : BOOL
VAR_INPUT
	fbMachineControlHMI	: ITF_MCHMIMachineControl_HMI_PrepScr_00_03;
END_VAR
this^.itfMachineControlHMI := fbMachineControlHMI;
END_METHOD

(*			
	RafalOS
	Rafał Osajda		14.11.2025		TC 4024.66
	Metoda przygotowywania danych dla HMI 
	W niej odbywa się odpytywanie właściego elementu przez łącznik
*)
METHOD PUBLIC PrepareDataForHMI : BOOL
VAR_INPUT
END_VAR
SUPER^.PrepareDataForHMI ();
END_METHOD

(*			
	RafalOS
	Rafał Osajda		19.11.2025		TC 4024.66
	Przygotowanie ramki pood tamke do wyświetlenia - tylko przygotowanie a nie przygotowanie danych do wyświetlenia
*)
METHOD PUBLIC PrepareForScreen : BOOL
VAR_INPUT
END_VAR
SUPER^.PrepareForScreen ();
END_METHOD

END_FUNCTION_BLOCK

// ---- POUs/06_MW_Washing/FB_MCHMIPrepareDataForScreen_00_04.TcPOU
(*			
	RafalOS
	Rafał Osajda		20.11.2025		TC 4024.66
	Moduł przygotowania danych dla Okna głównego w trybie mycia
*)
FUNCTION_BLOCK FB_MCHMIPrepareDataForScreen_00_04 EXTENDS FB_MCHMIPrepareDataForScreen IMPLEMENTS ITF_MCHMIPrepareDataForScreen
VAR
	itfMachineControlHMI	: ITF_MCHMIMachineControl_HMI_PrepScr_00_04;
	refstData				: REFERENCE TO ST_MCHMIPrepareScreen_00_04;
END_VAR

(*			
	RafalOS
	Rafał Osajda		19.11.2025		TC 4024.66
	Czyści danych przy zmienia ramki po poprzedniej ramce
*)
METHOD PUBLIC ClearAfterScreen : BOOL
VAR_INPUT
END_VAR
SUPER^.ClearAfterScreen ();
END_METHOD

METHOD PUBLIC LinkDataHMI_00_04 : BOOL
VAR_INPUT
	refstData				: REFERENCE TO ST_MCHMIPrepareScreen_00_04;
END_VAR
THIS^.refstData REF= refstData;
END_METHOD

METHOD PUBLIC LinkMachineControlHMI : BOOL
VAR_INPUT
	fbMachineControlHMI	: ITF_MCHMIMachineControl_HMI_PrepScr_00_04;
END_VAR
this^.itfMachineControlHMI := fbMachineControlHMI;
END_METHOD

(*			
	RafalOS
	Rafał Osajda		14.11.2025		TC 4024.66
	Metoda przygotowywania danych dla HMI 
	W niej odbywa się odpytywanie właściego elementu przez łącznik
*)
METHOD PUBLIC PrepareDataForHMI : BOOL
VAR_INPUT
END_VAR
SUPER^.PrepareDataForHMI ();
END_METHOD

(*			
	RafalOS
	Rafał Osajda		19.11.2025		TC 4024.66
	Przygotowanie ramki pood tamke do wyświetlenia - tylko przygotowanie a nie przygotowanie danych do wyświetlenia
*)
METHOD PUBLIC PrepareForScreen : BOOL
VAR_INPUT
END_VAR
SUPER^.PrepareForScreen ();
END_METHOD

END_FUNCTION_BLOCK

// ---- POUs/07_MW_Diagnostics/FB_MCHMIPrepareDataForScreen_00_05.TcPOU
(*			
	RafalOS
	Rafał Osajda		20.11.2025		TC 4024.66
	Moduł przygotowania danych dla Okna głównego w trybie diagnostyki
*)
FUNCTION_BLOCK FB_MCHMIPrepareDataForScreen_00_05 EXTENDS FB_MCHMIPrepareDataForScreen IMPLEMENTS ITF_MCHMIPrepareDataForScreen
VAR
	itfMachineControlHMI	: ITF_MCHMIMachineControl_HMI_PrepScr_00_05;
	refstData				: REFERENCE TO ST_MCHMIPrepareScreen_00_05;
END_VAR

(*			
	RafalOS
	Rafał Osajda		19.11.2025		TC 4024.66
	Czyści danych przy zmienia ramki po poprzedniej ramce
*)
METHOD PUBLIC ClearAfterScreen : BOOL
VAR_INPUT
END_VAR
SUPER^.ClearAfterScreen ();
END_METHOD

METHOD PUBLIC LinkDataHMI_00_05 : BOOL
VAR_INPUT
	refstData				: REFERENCE TO ST_MCHMIPrepareScreen_00_05;
END_VAR
THIS^.refstData REF= refstData;
END_METHOD

METHOD PUBLIC LinkMachineControlHMI : BOOL
VAR_INPUT
	fbMachineControlHMI	: ITF_MCHMIMachineControl_HMI_PrepScr_00_05;
END_VAR
this^.itfMachineControlHMI := fbMachineControlHMI;
END_METHOD

(*			
	RafalOS
	Rafał Osajda		14.11.2025		TC 4024.66
	Metoda przygotowywania danych dla HMI 
	W niej odbywa się odpytywanie właściego elementu przez łącznik
*)
METHOD PUBLIC PrepareDataForHMI : BOOL
VAR_INPUT
END_VAR
SUPER^.PrepareDataForHMI ();
END_METHOD

(*			
	RafalOS
	Rafał Osajda		19.11.2025		TC 4024.66
	Przygotowanie ramki pood tamke do wyświetlenia - tylko przygotowanie a nie przygotowanie danych do wyświetlenia
*)
METHOD PUBLIC PrepareForScreen : BOOL
VAR_INPUT
END_VAR
SUPER^.PrepareForScreen ();
END_METHOD

END_FUNCTION_BLOCK

// ---- POUs/08_Parameters/FB_MCHMIPrepareDataForScreen_01_XX.TcPOU
(*			
	RafalOS
	Rafał Osajda		20.11.2025		TC 4024.66
	Moduł przygotowania danych dla Okna parametrów we wsztsystkich trybach
*)
FUNCTION_BLOCK FB_MCHMIPrepareDataForScreen_01_XX EXTENDS FB_MCHMIPrepareDataForScreen IMPLEMENTS ITF_MCHMIPrepareDataForScreen
VAR
	itfMachineControlHMI	: ITF_MCHMIMachineControl_HMI_PrepScr_01_XX;
	refstData				: REFERENCE TO ST_MCHMIPrepareScreen_01_XX;
END_VAR

(*			
	RafalOS
	Rafał Osajda		19.11.2025		TC 4024.66
	Czyści danych przy zmienia ramki po poprzedniej ramce
*)
METHOD PUBLIC ClearAfterScreen : BOOL
VAR_INPUT
END_VAR
SUPER^.ClearAfterScreen ();
END_METHOD

METHOD PRIVATE CreateListName
VAR_INPUT
END_VAR
END_METHOD

METHOD PUBLIC LinkDataHMI_01_XX : BOOL
VAR_INPUT
	refstData				: REFERENCE TO ST_MCHMIPrepareScreen_01_XX;
END_VAR
THIS^.refstData REF= refstData;
END_METHOD

METHOD PUBLIC LinkMachineControlHMI : BOOL
VAR_INPUT
	fbMachineControlHMI	: ITF_MCHMIMachineControl_HMI_PrepScr_01_XX;
END_VAR
this^.itfMachineControlHMI := fbMachineControlHMI;
END_METHOD

(*			
	RafalOS
	Rafał Osajda		14.11.2025		TC 4024.66
	Metoda przygotowywania danych dla HMI 
	W niej odbywa się odpytywanie właściego elementu przez łącznik
*)
METHOD PUBLIC PrepareDataForHMI : BOOL
VAR_INPUT
END_VAR

IF (THIS^.refstHMICommonData.bChangePage) THEN
	THIS^.CreateListName ();
END_IF





SUPER^.PrepareDataForHMI ();
END_METHOD

(*			
	RafalOS
	Rafał Osajda		19.11.2025		TC 4024.66
	Przygotowanie ramki pood tamke do wyświetlenia - tylko przygotowanie a nie przygotowanie danych do wyświetlenia
*)
METHOD PUBLIC PrepareForScreen : BOOL
VAR_INPUT
END_VAR
SUPER^.PrepareForScreen ();
END_METHOD

END_FUNCTION_BLOCK

// ---- POUs/09_Recipe/FB_MCHMIPrepareDataForScreen_02_XX.TcPOU
(*			
	RafalOS
	Rafał Osajda		20.11.2025		TC 4024.66
	Moduł przygotowania danych dla Okna receptur we wszsytkich trybach
*)
FUNCTION_BLOCK FB_MCHMIPrepareDataForScreen_02_XX EXTENDS FB_MCHMIPrepareDataForScreen IMPLEMENTS ITF_MCHMIPrepareDataForScreen
VAR
	itfMachineControlHMI	: ITF_MCHMIMachineControl_HMI_PrepScr_02_XX;
	refstData				: REFERENCE TO ST_MCHMIPrepareScreen_02_XX;
	stTitleRecipe			: ST_BaseLabel;
	stSourceRecipe			: ST_BaseLabel;
	stTitleTemplate			: ST_BaseLabel;
	stSourceTemplate		: ST_BaseLabel;
	stDeleteRecipe			: ST_BaseLabel;
END_VAR

(*			
	RafalOS
	Rafał Osajda		19.11.2025		TC 4024.66
	Czyści danych przy zmienia ramki po poprzedniej ramce
*)
METHOD PUBLIC ClearAfterScreen : BOOL
VAR_INPUT
END_VAR
SUPER^.ClearAfterScreen ();
END_METHOD

METHOD PRIVATE CreateListName : BOOL
VAR
	stNameList		: ST_BaseRecipeList;	
	iI				: INT;
END_VAR
THIS^.refstData.bRefreshList := FALSE;
stNameList := THIS^.itfMachineControlHMI.GetListOfNameRecipe ();
THIS^.refstData.iNumberOfRecipe := stNameList.iNumber;
FOR iI := 1 TO stNameList.iNumber DO
	THIS^.refstData.arrNameListRecipe [iI] := GetTextFromLabelForActiveLocation (
											stLabel := stNameList.arrName [iI]
										);
END_FOR
IF (stNameList.iNumber = 0) THEN
	THIS^.refstData.bSelectedNameRow := FALSE;
	THIS^.refstData.iSelectedNameRow := 0;
	MEMSET (
		destAddr := ADR (THIS^.refstData.arrNameListRecipe),
		fillByte := 0,
		n := SIZEOF (THIS^.refstData.arrNameListRecipe)
	);
END_IF
stNameList := THIS^.itfMachineControlHMI.GetListOfNameTemplate ();
THIS^.refstData.iNumberOfTemplate := stNameList.iNumber;
FOR iI := 1 TO stNameList.iNumber DO
	THIS^.refstData.arrNameListTemplate [iI] := GetTextFromLabelForActiveLocation (
													stLabel := stNameList.arrName [iI]
												);
END_FOR
END_METHOD

METHOD PUBLIC LinkDataHMI_02_XX : BOOL
VAR_INPUT
	refstData				: REFERENCE TO ST_MCHMIPrepareScreen_02_XX;
END_VAR
THIS^.refstData REF= refstData;
END_METHOD

METHOD PUBLIC LinkMachineControlHMI : BOOL
VAR_INPUT
	fbMachineControlHMI	: ITF_MCHMIMachineControl_HMI_PrepScr_02_XX;
END_VAR
this^.itfMachineControlHMI := fbMachineControlHMI;
END_METHOD

METHOD PRIVATE PrepareDataAddRecipe : BOOL
VAR_INST
	rtAddRecipeFromTemplate		: R_TRIG;
	rtAddRecipeFromRecipe		: R_TRIG;
END_VAR

VAR
	btmpAddRecipe: BOOL;
END_VAR
	(*	Dodawanie Receptury	*)
rtAddRecipeFromTemplate (CLK := refstData.stAddRecipe.bNewRecipeFromTemplate);
rtAddRecipeFromRecipe (CLK := refstData.stAddRecipe.bNewRecipeFromRecipe);

IF (rtAddRecipeFromTemplate.Q) THEN
	refstData.stAddRecipe.arrListOfName := refstData.arrNameListTemplate;
	refstData.stAddRecipe.iNumberOfNames := refstData.iNumberOfTemplate;
	refstData.stAddRecipe.iSelectedName := -1;
	THIS^.SetText (eLocation := E_BaseLocation.pl, wsDescription := "");
	THIS^.SetText (eLocation := E_BaseLocation.en, wsDescription := "");
	THIS^.SetText (eLocation := E_BaseLocation.de, wsDescription := "");
	refstData.stAddRecipe.stNewNames := THIS^.GetTexts ();
	refstData.stAddRecipe.wsTitle := THIS^.GetTextFromLabelForActiveLocation (
										stLabel := THIS^.stTitleTemplate
									);
	refstData.stAddRecipe.wsSource := THIS^.GetTextFromLabelForActiveLocation (
										stLabel := THIS^.stSourceTemplate
									);
END_IF
IF (rtAddRecipeFromRecipe.Q) THEN
	refstData.stAddRecipe.arrListOfName := refstData.arrNameListRecipe;
	refstData.stAddRecipe.iNumberOfNames := refstData.iNumberOfRecipe;
	refstData.stAddRecipe.iSelectedName := refstData.iSelectedNameRow;
	THIS^.SetText (eLocation := E_BaseLocation.pl, wsDescription := "");
	THIS^.SetText (eLocation := E_BaseLocation.en, wsDescription := "");
	THIS^.SetText (eLocation := E_BaseLocation.de, wsDescription := "");
	refstData.stAddRecipe.stNewNames := THIS^.GetTexts ();
	refstData.stAddRecipe.wsTitle := THIS^.GetTextFromLabelForActiveLocation (
										stLabel := THIS^.stTitleRecipe
									);
	refstData.stAddRecipe.wsSource := THIS^.GetTextFromLabelForActiveLocation (
										stLabel := THIS^.stSourceRecipe
									);
END_IF
	
IF (refstData.stAddRecipe.bOk AND refstData.stAddRecipe.bNewRecipeFromTemplate) THEN
	IF (refstData.stAddRecipe.bSelectedRow AND refstData.stAddRecipe.stNewNames.arrText [1] <> "") THEN
		THIS^.itfMachineControlHMI.AddRecipeFromTemplate (
			uiNumberTemplates := TO_UINT (refstData.stAddRecipe.iSelectedName),
			stTexts := refstData.stAddRecipe.stNewNames
		);
		btmpAddRecipe := TRUE;
	ELSE
		refstData.stAddRecipe.bCancel := TRUE;
	END_IF
END_IF
IF (refstData.stAddRecipe.bOk AND refstData.stAddRecipe.bNewRecipeFromRecipe) THEN
	IF (refstData.stAddRecipe.bSelectedRow AND refstData.stAddRecipe.arrListOfName [1] <> "") THEN
		THIS^.itfMachineControlHMI.AddRecipeFromRecipe (
			uiNumberRecipe := TO_UINT (refstData.stAddRecipe.iSelectedName),
			stTexts := refstData.stAddRecipe.stNewNames
		);
		btmpAddRecipe := TRUE;
	ELSE
		refstData.stAddRecipe.bCancel := TRUE;
	END_IF
END_IF
IF (btmpAddRecipe) THEN
	btmpAddRecipe := FALSE;
	refstData.stAddRecipe.bOk := FALSE;
	THIS^.refstData.bRefreshList := TRUE;
	refstData.iSelectedNameRow := TO_INT (THIS^.itfMachineControlHMI.GetNumberOfRecipe ());
	refstData.bSelectedNameRow := TRUE;
	refstData.stAddRecipe.bNewRecipeFromTemplate := FALSE;
	refstData.stAddRecipe.bNewRecipeFromRecipe := FALSE;
END_IF
IF (refstData.stAddRecipe.bCancel) THEN
	refstData.stAddRecipe.bCancel := FALSE;
	refstData.stAddRecipe.bOk := FALSE;
	refstData.stAddRecipe.bNewRecipeFromTemplate := FALSE;
	refstData.stAddRecipe.bNewRecipeFromRecipe := FALSE;
END_IF
END_METHOD

METHOD PRIVATE PrepareDataChangePage : BOOL
VAR_INPUT
END_VAR
THIS^.refstData.stIngredientList.stList.iSelectedRow := 0;
THIS^.refstData.stIngredientList.stList.bSelectedRow := FALSE;
THIS^.refstData.stIngredientList.iStartIndex := THIS^.refstData.stIngredientList.iActualPage * 
												GVL_MCHMIConstans.NUMBER_INDEGRIEND_ON_PAGE + 1 - 10;
THIS^.PrepareDataFillIngredientTable (
	iRecipe		:= THIS^.refstData.iSelectedNameRow,
	iStartIndex	:= THIS^.refstData.stIngredientList.iStartIndex,
);
END_METHOD

METHOD PRIVATE PrepareDataDeleteRacipe : BOOL
VAR_INST
	rtDelete		: r_trig;
	
END_VAR
rtDelete (CLK := THIS^.refstData.stDeleteRecipe.bDeleteRecipe);

IF (rtDelete.Q) THEN
	THIS^.refstData.stDeleteRecipe.wsDescription := THIS^.GetTextFromLabelForActiveLocation (
														stLabel := THIS^.stDeleteRecipe
													);
	THIS^.refstData.stDeleteRecipe.wsNameRecipe := THIS^.refstData.arrNameListRecipe [THIS^.refstData.iSelectedNameRow];
END_IF

IF (THIS^.refstData.stDeleteRecipe.bOK AND THIS^.refstData.stDeleteRecipe.bDeleteRecipe) THEN
	THIS^.refstData.stDeleteRecipe.bOK := FALSE;
	THIS^.refstData.stDeleteRecipe.bDeleteRecipe := FALSE;
	IF (THIS^.refstData.iSelectedNameRow = TO_INT (THIS^.itfMachineControlHMI.GetNumberOfChoosen ())) THEN
		THIS^.itfMachineControlHMI.ClearChosen ();
	END_IF
	THIS^.itfMachineControlHMI.DeleteRecipe (uiNumber := TO_UINT (THIS^.refstData.iSelectedNameRow));
	THIS^.refstData.bRefreshList := TRUE;
	THIS^.refstData.iSelectedNameRow := -1;
	THIS^.refstData.iSelectedNameRowPrev := -1;
	THIS^.refstData.bSelectedNameRow := FALSE;
END_IF
IF (THIS^.refstData.stDeleteRecipe.bCancel AND THIS^.refstData.stDeleteRecipe.bDeleteRecipe) THEN
	THIS^.refstData.stDeleteRecipe.bCancel := FALSE;
	THIS^.refstData.stDeleteRecipe.bDeleteRecipe := FALSE;
END_IF
END_METHOD

METHOD PRIVATE PrepareDataFillIngredientTable : BOOL
VAR_INPUT
	iRecipe			: INT;	//numer receptury z której bierzemy składniki
	iStartIndex		: INT;	//numer startowy składnika
END_VAR
VAR
	arrtmpResultPage	: ARRAY [0..GVL_MCHMIConstans.NUMBER_INDEGRIEND_ON_PAGE] OF ST_BaseDescriptor;
	iI					: INT;
	
END_VAR
THIS^.itfMachineControlHMI.GetIngredientRange (
	iRecipe		:= iRecipe,
	iStartIndex	:= iStartIndex,
	iCount		:= GVL_MCHMIConstans.NUMBER_INDEGRIEND_ON_PAGE + 1,	//liczba musi byc równa ilości pol w tablicy przekazywanej
	arrOut		:= arrtmpResultPage,
	iNumberOfFilledData => THIS^.refstData.stIngredientList.iNumberRowOnPage
);
FOR iI := 1 TO GVL_MCHMIConstans.NUMBER_INDEGRIEND_ON_PAGE DO
	THIS^.refstData.stIngredientList.stList.arrRow [iI].wsText :=
		THIS^.GetTextFromLabelForActiveLocation (stLabel := arrtmpResultPage [iI].stTexts);
	THIS^.refstData.stIngredientList.stList.arrRow [iI].rValue := arrtmpResultPage [iI].rValue;
	THIS^.refstData.stIngredientList.stList.arrRow [iI].rMin := arrtmpResultPage [iI].rMin;
	THIS^.refstData.stIngredientList.stList.arrRow [iI].rMax := arrtmpResultPage [iI].rMax;
	THIS^.refstData.stIngredientList.stList.arrRow [iI].rDefaultValue := arrtmpResultPage [iI].rDefaultValue;
	THIS^.refstData.stIngredientList.stList.arrRow [iI].sUnit := arrtmpResultPage [iI].sUnit;
END_FOR
END_METHOD

(*			
	RafalOS
	Rafał Osajda		05.12.2025		TC 4024.66
	Przygotowanie danych przy pierwszym wejściu do okienka
*)
METHOD PRIVATE PrepareDataFirstPageIngediends : BOOL
VAR_INPUT
END_VAR
THIS^.refstData.stIngredientList.iActualPage := 1;
THIS^.refstData.stIngredientList.stList.iSelectedRow := 0;
THIS^.refstData.stIngredientList.stList.iSelectedRowPrev := 0;
THIS^.refstData.stIngredientList.stList.bSelectedRow := FALSE;
THIS^.refstData.stIngredientList.iStartIndex := 1;
THIS^.refstData.stIngredientList.iTotal := TO_INT (
		THIS^.itfMachineControlHMI.GetNumberIngredientOfRecipe (
			uiNumber := TO_UINT (THIS^.refstData.iSelectedNameRow)
		));
THIS^.refstData.stIngredientList.iNumberOfPage := 
	(THIS^.refstData.stIngredientList.iTotal + GVL_MCHMIConstans.NUMBER_INDEGRIEND_ON_PAGE -1 ) / 
		GVL_MCHMIConstans.NUMBER_INDEGRIEND_ON_PAGE;
THIS^.PrepareDataFillIngredientTable (
	iRecipe		:= THIS^.refstData.iSelectedNameRow,
	iStartIndex	:= THIS^.refstData.stIngredientList.iStartIndex,
);
END_METHOD

(*			
	RafalOS
	Rafał Osajda		14.11.2025		TC 4024.66
	Metoda przygotowywania danych dla HMI 
	W niej odbywa się odpytywanie właściego elementu przez łącznik
*)
METHOD PUBLIC PrepareDataForHMI : BOOL
VAR
	btmpAddRecipe		: BOOL;
	arrtmpResultPage	: ARRAY [0..GVL_MCHMIConstans.NUMBER_INDEGRIEND_ON_PAGE] OF ST_BaseDescriptor;
	iI: INT;
END_VAR
	(*	Lista receptur	*)

IF (THIS^.refstHMICommonData.bChangePage OR THIS^.refstData.bRefreshList) THEN
	THIS^.CreateListName ();
END_IF
	(*	Obsługa przycisków zarządzania recepturami	*)
	
THIS^.refstData.bVisibleButtonAddFromRecipe := THIS^.refstData.bSelectedNameRow;
THIS^.refstData.bVisibleButtonAddFromTemplate := THIS^.refstData.iNumberOfTemplate > 0;
THIS^.refstData.bVisibleButtonDelete := THIS^.refstData.bSelectedNameRow;
THIS^.refstData.bVsibleButtonEditIngredient := THIS^.refstData.bSelectedNameRow;
THIS^.refstData.bVisibleButtonChoose := THIS^.refstData.bSelectedNameRow AND 
										TO_INT (THIS^.itfMachineControlHMI.GetNumberOfChoosen ()) <> THIS^.refstData.iSelectedNameRow; //and not test czy receputa wybrana;
	
THIS^.PrepareDataAddRecipe ();
THIS^.PrepareDataDeleteRacipe ();

	(*	Lista składników receptury	*)

IF (THIS^.refstData.iSelectedNameRow <> THIS^.refstData.iSelectedNameRowPrev AND THIS^.refstData.bSelectedNameRow) THEN
	THIS^.refstData.iSelectedNameRowPrev := THIS^.refstData.iSelectedNameRow;
	THIS^.PrepareDataFirstPageIngediends ();	//przygotowanie pierwszej strony listy przy zmianie receptury
END_IF
IF (THIS^.refstData.stIngredientList.iActualPage <> THIS^.refstData.stIngredientList.iPreviewPage) THEN
	THIS^.refstData.stIngredientList.iPreviewPage := THIS^.refstData.stIngredientList.iActualPage;
	THIS^.PrepareDataChangePage (); //zmiana strony
END_IF
IF (THIS^.refstData.stIngredientList.bRefresh) THEN //odświerzenie listy składników
	THIS^.PrepareDataFillIngredientTable (
		iRecipe		:= THIS^.refstData.iSelectedNameRow,
		iStartIndex	:= THIS^.refstData.stIngredientList.iStartIndex,
	);	
END_IF
IF ( (THIS^.refstData.stIngredientList.stList.iSelectedRow <> THIS^.refstData.stIngredientList.stList.iSelectedRowPrev OR
	THIS^.refstData.stIngredientList.bRefresh) AND
	THIS^.refstData.bSelectedNameRow) THEN
	THIS^.refstData.stIngredientList.stList.iSelectedRowPrev := THIS^.refstData.stIngredientList.stList.iSelectedRow;
	THIS^.refstData.stIngredientList.bRefresh := FALSE;
	THIS^.PrepareDataSelectedIngeriend ();
END_IF
	(*	Wybranie receptury	*)
IF (THIS^.refstData.bSelectRecipe) THEN
	THIS^.refstData.bSelectRecipe := FALSE;
	THIS^.itfMachineControlHMI.SelectRecipe (
		uiRecipe := TO_UINT (THIS^.refstData.iSelectedNameRow)
	);
	THIS^.refstHMICommonData.stRecipeInformation.bNewSelectedRecipe := TRUE;
END_IF

THIS^.refstData.stIngredientList.stChossenRow.bVisibleSave := THIS^.refstData.stIngredientList.stChossenRow.rValue <> 
										THIS^.refstData.stIngredientList.stChossenRow.rValueOld;
THIS^.refstData.stIngredientList.stChossenRow.bVisibleSetDefault := THIS^.refstData.stIngredientList.stChossenRow.rValue <> 
										THIS^.refstData.stIngredientList.stChossenRow.rDefaultValue;
THIS^.refstData.stIngredientList.stChossenRow.bVisibleCancel := THIS^.refstData.stIngredientList.stChossenRow.rValue <> 
										THIS^.refstData.stIngredientList.stChossenRow.rValueOld;

IF (THIS^.refstData.stIngredientList.stChossenRow.bSave) THEN
	THIS^.refstData.stIngredientList.stChossenRow.bSave := FALSE;
	THIS^.itfMachineControlHMI.SetIngredientValue (
		iRecipe := THIS^.refstData.iSelectedNameRow,
		iIngredient := THIS^.refstData.stIngredientList.stChossenRow.iID,
		rValue := THIS^.refstData.stIngredientList.stChossenRow.rValue
	);
	THIS^.itfMachineControlHMI.ClearChosen ();
	THIS^.refstData.stIngredientList.bRefresh := TRUE;
END_IF
IF (THIS^.refstData.stIngredientList.stChossenRow.bSetDefault) THEN
	THIS^.refstData.stIngredientList.stChossenRow.bSetDefault := FALSE;
	THIS^.refstData.stIngredientList.stChossenRow.rValue := THIS^.refstData.stIngredientList.stChossenRow.rDefaultValue;
END_IF
IF (THIS^.refstData.stIngredientList.stChossenRow.bCancel) THEN
	THIS^.refstData.stIngredientList.stChossenRow.bCancel := FALSE;
	THIS^.refstData.stIngredientList.stChossenRow.rValue := THIS^.refstData.stIngredientList.stChossenRow.rValueOld;
END_IF



	(*	Zewnętrzna obsługa wyświetlania 	*)
SUPER^.PrepareDataForHMI ();
END_METHOD

(*			
	RafalOS
	Rafał Osajda		05.12.2025		TC 4024.66
	Wyświetl dane dla wybranego deskryptora
*)
METHOD PRIVATE PrepareDataSelectedIngeriend : BOOL
VAR
	iIndex		: INT;
	stResult	: ST_BaseDescriptor;
END_VAR
iIndex := THIS^.refstData.stIngredientList.iActualPage * GVL_MCHMIConstans.NUMBER_INDEGRIEND_ON_PAGE 
				- 10 + THIS^.refstData.stIngredientList.stList.iSelectedRow;

stResult := THIS^.itfMachineControlHMI.GetIngredientFromRecipe (
				uiNumberOfRecipe := TO_UINT (THIS^.refstData.iSelectedNameRow),
				uiNumberOfIngredient := TO_UINT (iIndex)
			);

THIS^.refstData.stIngredientList.stChossenRow.wsText := THIS^.GetTextFromLabelForActiveLocation (
										stLabel := stResult.stTexts
									);
THIS^.refstData.stIngredientList.stChossenRow.rValue := stResult.rValue;
THIS^.refstData.stIngredientList.stChossenRow.rValueOld := stResult.rValue;
THIS^.refstData.stIngredientList.stChossenRow.rMin := stResult.rMin;
THIS^.refstData.stIngredientList.stChossenRow.rMax := stResult.rMax;
THIS^.refstData.stIngredientList.stChossenRow.rDefaultValue := stResult.rDefaultValue;
THIS^.refstData.stIngredientList.stChossenRow.sUnit := stResult.sUnit;
THIS^.refstData.stIngredientList.stChossenRow.iID := iIndex;
END_METHOD

(*			
	RafalOS
	Rafał Osajda		19.11.2025		TC 4024.66
	Przygotowanie ramki pood tamke do wyświetlenia - tylko przygotowanie a nie przygotowanie danych do wyświetlenia
*)
METHOD PUBLIC PrepareForScreen : BOOL
VAR_INPUT
END_VAR
THIS^.SetText (eLocation := E_BaseLocation.pl, wsDescription := "Utwórz recepturę z szablonu");
THIS^.SetText (eLocation := E_BaseLocation.en, wsDescription := "");
THIS^.SetText (eLocation := E_BaseLocation.de, wsDescription := "");
THIS^.stTitleRecipe := THIS^.GetTexts ();
THIS^.SetText (eLocation := E_BaseLocation.pl, wsDescription := "Wybierz szablon");
THIS^.SetText (eLocation := E_BaseLocation.en, wsDescription := "");
THIS^.SetText (eLocation := E_BaseLocation.de, wsDescription := "");
THIS^.stSourceRecipe := THIS^.GetTexts ();

THIS^.SetText (eLocation := E_BaseLocation.pl, wsDescription := "Utwórz recepturę z receptury");
THIS^.SetText (eLocation := E_BaseLocation.en, wsDescription := "");
THIS^.SetText (eLocation := E_BaseLocation.de, wsDescription := "");
THIS^.stTitleTemplate := THIS^.GetTexts ();
THIS^.SetText (eLocation := E_BaseLocation.pl, wsDescription := "Wybierz recepturę");
THIS^.SetText (eLocation := E_BaseLocation.en, wsDescription := "");
THIS^.SetText (eLocation := E_BaseLocation.de, wsDescription := "");
THIS^.stSourceTemplate := THIS^.GetTexts ();

THIS^.SetText (eLocation := E_BaseLocation.pl, wsDescription := "Czy napewno usunąć recepturę");
THIS^.SetText (eLocation := E_BaseLocation.en, wsDescription := "");
THIS^.SetText (eLocation := E_BaseLocation.de, wsDescription := "");
THIS^.stDeleteRecipe := THIS^.GetTexts ();


SUPER^.PrepareForScreen ();
END_METHOD

END_FUNCTION_BLOCK

// ---- POUs/10_Alarm/FB_MCHMIPrepareDataForScreen_03_XX.TcPOU
(*			
	RafalOS
	Rafał Osajda		20.11.2025		TC 4024.66
	Moduł przygotowania danych dla Okna zdarzeń we wszystkich trybach
*)
FUNCTION_BLOCK FB_MCHMIPrepareDataForScreen_03_XX EXTENDS FB_MCHMIPrepareDataForScreen IMPLEMENTS ITF_MCHMIPrepareDataForScreen
VAR
	itfMachineControlHMI	: ITF_MCHMIMachineControl_HMI_PrepScr_03_XX;
	refstData				: REFERENCE TO ST_MCHMIPrepareScreen_03_XX;
END_VAR

(*			
	RafalOS
	Rafał Osajda		19.11.2025		TC 4024.66
	Czyści danych przy zmienia ramki po poprzedniej ramce
*)
METHOD PUBLIC ClearAfterScreen : BOOL
VAR_INPUT
END_VAR
SUPER^.ClearAfterScreen ();
END_METHOD

METHOD PUBLIC LinkDataHMI_03_XX : BOOL
VAR_INPUT
	refstData				: REFERENCE TO ST_MCHMIPrepareScreen_03_XX;
END_VAR
THIS^.refstData REF= refstData;
END_METHOD

METHOD PUBLIC LinkMachineControlHMI : BOOL
VAR_INPUT
	fbMachineControlHMI	: ITF_MCHMIMachineControl_HMI_PrepScr_03_XX;
END_VAR
this^.itfMachineControlHMI := fbMachineControlHMI;
END_METHOD

(*			
	RafalOS
	Rafał Osajda		14.11.2025		TC 4024.66
	Metoda przygotowywania danych dla HMI 
	W niej odbywa się odpytywanie właściego elementu przez łącznik
*)
METHOD PUBLIC PrepareDataForHMI : BOOL
VAR_INPUT
END_VAR
SUPER^.PrepareDataForHMI ();
END_METHOD

(*			
	RafalOS
	Rafał Osajda		19.11.2025		TC 4024.66
	Przygotowanie ramki pood tamke do wyświetlenia - tylko przygotowanie a nie przygotowanie danych do wyświetlenia
*)
METHOD PUBLIC PrepareForScreen : BOOL
VAR_INPUT
END_VAR
SUPER^.PrepareForScreen ();
END_METHOD

END_FUNCTION_BLOCK

// ---- POUs/11_ChangeMode/FB_MCHMIPrepareDataForScreen_04_XX.TcPOU
(*			
	RafalOS
	Rafał Osajda		20.11.2025		TC 4024.66
	Moduł przygotowania danych dla Okna zmiany trybu we wszystkich trybach
*)
FUNCTION_BLOCK FB_MCHMIPrepareDataForScreen_04_XX EXTENDS FB_MCHMIPrepareDataForScreen IMPLEMENTS ITF_MCHMIPrepareDataForScreen
VAR
	itfMachineControlHMI	: ITF_MCHMIMachineControl_HMI_PrepScr_04_XX;
	refstData				: REFERENCE TO ST_MCHMIPrepareScreen_04_XX;
END_VAR

(*			
	RafalOS
	Rafał Osajda		19.11.2025		TC 4024.66
	Czyści danych przy zmienia ramki po poprzedniej ramce
*)
METHOD PUBLIC ClearAfterScreen : BOOL
VAR_INPUT
END_VAR
SUPER^.ClearAfterScreen ();
END_METHOD

METHOD PUBLIC LinkDataHMI_04_XX : BOOL
VAR_INPUT
	refstData				: REFERENCE TO ST_MCHMIPrepareScreen_04_XX;
END_VAR
THIS^.refstData REF= refstData;
END_METHOD

METHOD PUBLIC LinkMachineControlHMI : BOOL
VAR_INPUT
	fbMachineControlHMI	: ITF_MCHMIMachineControl_HMI_PrepScr_04_XX;
END_VAR
this^.itfMachineControlHMI := fbMachineControlHMI;
END_METHOD

(*			
	RafalOS
	Rafał Osajda		14.11.2025		TC 4024.66
	Metoda przygotowywania danych dla HMI 
	W niej odbywa się odpytywanie właściego elementu przez łącznik
*)
METHOD PUBLIC PrepareDataForHMI : BOOL
VAR_INST
	etmpMode					: E_BaseMachineMode := E_BaseMachineMode.NotAllowed;
END_VAR
VAR
	iJ							: INT;
	iActiveMode					: E_BaseMachineMode;
	etmpCmdChangeMode			: E_SaMCommandChangeMode;
END_VAR
THIS^.refstData.wsActualMode := THIS^.GetTextFromLabelForActiveLocation (THIS^.itfMachineControlHMI.GetActiveModeName ());
THIS^.refstData.eActualMode := THIS^.itfMachineControlHMI.GetActiveMode ();


	(*	Przygotowanie ifnormacji dla zmiany trybu	*)

IF (THIS^.refstHMICommonData.bChangePage OR etmpMode <> THIS^.refstData.eActualMode) THEN
	etmpMode := THIS^.refstData.eActualMode;
	THIS^.refstData.iNumberModeToDisplay := 0;
	iActiveMode := THIS^.itfMachineControlHMI.GetActiveMode ();
	FOR iJ := 1 TO GVL_SaMConstans.NUMBER_OF_MODES DO
		IF (THIS^.itfMachineControlHMI.IsModeEnabled (iMode := iJ) AND iJ <> iActiveMode) THEN
			THIS^.refstData.arrNamesOfMode [THIS^.refstData.iNumberModeToDisplay].wsDescription := 
				THIS^.GetTextFromLabelForActiveLocation (stLabel := THIS^.itfMachineControlHMI.GetModeName (iMode := iJ));
			THIS^.refstData.arrNamesOfMode [THIS^.refstData.iNumberModeToDisplay].iNumber := iJ;
			THIS^.refstData.iNumberModeToDisplay := THIS^.refstData.iNumberModeToDisplay + 1;
			THIS^.refstData.iSelectedMode := -1;
		END_IF
	END_FOR
END_IF
IF (THIS^.refstData.bChangeMode AND THIS^.refstData.bSelectedRow) THEN
	THIS^.refstData.bChangeMode := FALSE;
	//polecenie zmiany trybu 
	CASE THIS^.refstData.arrNamesOfMode [THIS^.refstData.iSelectedMode].iNumber OF
	E_SaMCommandChangeMode.Production : etmpCmdChangeMode := E_SaMCommandChangeMode.Production;
	E_SaMCommandChangeMode.Maintenance : etmpCmdChangeMode := E_SaMCommandChangeMode.Maintenance;
	E_SaMCommandChangeMode.Manual : etmpCmdChangeMode := E_SaMCommandChangeMode.Manual;
	E_SaMCommandChangeMode.Washing : etmpCmdChangeMode := E_SaMCommandChangeMode.Washing;
	E_SaMCommandChangeMode.Diagnostisc : etmpCmdChangeMode := E_SaMCommandChangeMode.Diagnostisc;
	END_CASE
	THIS^.itfMachineControlHMI.SetCmdChangeMode (eCmdNumber := etmpCmdChangeMode);
	THIS^.refstData.iSelectedMode := -1;
END_IF



SUPER^.PrepareDataForHMI ();
END_METHOD

(*			
	RafalOS
	Rafał Osajda		19.11.2025		TC 4024.66
	Przygotowanie ramki pood tamke do wyświetlenia - tylko przygotowanie a nie przygotowanie danych do wyświetlenia
*)
METHOD PUBLIC PrepareForScreen : BOOL
VAR_INPUT
END_VAR
SUPER^.PrepareForScreen ();
END_METHOD

END_FUNCTION_BLOCK

// ---- POUs/12_Statistics/FB_MCHMIPrepareDataForScreen_05_XX.TcPOU
(*			
	RafalOS
	Rafał Osajda		20.11.2025		TC 4024.66
	Moduł przygotowania danych dla Okna statystyk we wszsytkich trybach
*)
FUNCTION_BLOCK FB_MCHMIPrepareDataForScreen_05_XX EXTENDS FB_MCHMIPrepareDataForScreen IMPLEMENTS ITF_MCHMIPrepareDataForScreen
VAR
	itfMachineControlHMI	: ITF_MCHMIMachineControl_HMI_PrepScr_05_XX;
	refstData				: REFERENCE TO ST_MCHMIPrepareScreen_05_XX;
END_VAR

(*			
	RafalOS
	Rafał Osajda		19.11.2025		TC 4024.66
	Czyści danych przy zmienia ramki po poprzedniej ramce
*)
METHOD PUBLIC ClearAfterScreen : BOOL
VAR_INPUT
END_VAR
SUPER^.ClearAfterScreen ();
END_METHOD

METHOD PUBLIC LinkDataHMI_05_XX : BOOL
VAR_INPUT
	refstData				: REFERENCE TO ST_MCHMIPrepareScreen_05_XX;
END_VAR
THIS^.refstData REF= refstData;
END_METHOD

METHOD PUBLIC LinkMachineControlHMI : BOOL
VAR_INPUT
	fbMachineControlHMI	: ITF_MCHMIMachineControl_HMI_PrepScr_05_XX;
END_VAR
this^.itfMachineControlHMI := fbMachineControlHMI;
END_METHOD

(*			
	RafalOS
	Rafał Osajda		14.11.2025		TC 4024.66
	Metoda przygotowywania danych dla HMI 
	W niej odbywa się odpytywanie właściego elementu przez łącznik
*)
METHOD PUBLIC PrepareDataForHMI : BOOL
VAR_INPUT
END_VAR
SUPER^.PrepareDataForHMI ();
END_METHOD

(*			
	RafalOS
	Rafał Osajda		19.11.2025		TC 4024.66
	Przygotowanie ramki pood tamke do wyświetlenia - tylko przygotowanie a nie przygotowanie danych do wyświetlenia
*)
METHOD PUBLIC PrepareForScreen : BOOL
VAR_INPUT
END_VAR
SUPER^.PrepareForScreen ();
END_METHOD

END_FUNCTION_BLOCK

// ---- POUs/13_StateDiagram/FB_MCHMIPrepareDataForScreen_06_XX.TcPOU
(*			
	RafalOS
	Rafał Osajda		20.11.2025		TC 4024.66
	Moduł przygotowania danych dla Okna diagramu we wszystkich trybach
*)
FUNCTION_BLOCK FB_MCHMIPrepareDataForScreen_06_XX EXTENDS FB_MCHMIPrepareDataForScreen IMPLEMENTS ITF_MCHMIPrepareDataForScreen
VAR
	itfMachineControlHMI	: ITF_MCHMIMachineControl_HMI_PrepScr_06_XX;
	refstData				: REFERENCE TO ST_MCHMIPrepareScreen_06_XX;

	eActiveMode				: E_BaseMachineMode;
	
END_VAR

(*			
	RafalOS
	Rafał Osajda		19.11.2025		TC 4024.66
	Czyści danych przy zmienia ramki po poprzedniej ramce
*)
METHOD PUBLIC ClearAfterScreen : BOOL
VAR_INPUT
END_VAR
SUPER^.ClearAfterScreen ();
END_METHOD

METHOD PUBLIC LinkDataHMI_06_XX : BOOL
VAR_INPUT
	refstData				: REFERENCE TO ST_MCHMIPrepareScreen_06_XX;
END_VAR
THIS^.refstData REF= refstData;
END_METHOD

METHOD PUBLIC LinkMachineControlHMI : BOOL
VAR_INPUT
	fbMachineControlHMI	: ITF_MCHMIMachineControl_HMI_PrepScr_06_XX;
END_VAR
this^.itfMachineControlHMI := fbMachineControlHMI;
END_METHOD

(*			
	RafalOS
	Rafał Osajda		24.11.2025		TC 4024.66
	Obsługa przycisków zmiany stanu w diagramie
*)
METHOD PRIVATE PrepareButtonChangeState
VAR
	iI: INT;
END_VAR
FOR iI := 1 TO GVL_SaMConstans.NUMBER_OF_COMMAND_CHANGE_STATES DO
	IF (THIS^.refstData.arrCmdChangeState [iI].bPushed) THEN
		THIS^.refstData.arrCmdChangeState [iI].bPushed := FALSE;
		CASE iI OF
		E_SaMCommandChangeState.Abort 		: THIS^.itfMachineControlHMI.SetCmdChangeState (eCmdNumber := E_SaMCommandChangeState.Abort);
		E_SaMCommandChangeState.Clear 		: THIS^.itfMachineControlHMI.SetCmdChangeState (eCmdNumber := E_SaMCommandChangeState.Clear);
		E_SaMCommandChangeState.Reset		: THIS^.itfMachineControlHMI.SetCmdChangeState (eCmdNumber := E_SaMCommandChangeState.Reset);
		E_SaMCommandChangeState.Start		: THIS^.itfMachineControlHMI.SetCmdChangeState (eCmdNumber := E_SaMCommandChangeState.Start);
		E_SaMCommandChangeState.Stop		: THIS^.itfMachineControlHMI.SetCmdChangeState (eCmdNumber := E_SaMCommandChangeState.Stop);
		E_SaMCommandChangeState.Hold		: THIS^.itfMachineControlHMI.SetCmdChangeState (eCmdNumber := E_SaMCommandChangeState.Hold);
		E_SaMCommandChangeState.Unhold		: THIS^.itfMachineControlHMI.SetCmdChangeState (eCmdNumber := E_SaMCommandChangeState.Unhold);
		E_SaMCommandChangeState.Suspend		: THIS^.itfMachineControlHMI.SetCmdChangeState (eCmdNumber := E_SaMCommandChangeState.Suspend);
		E_SaMCommandChangeState.Unsuspend	: THIS^.itfMachineControlHMI.SetCmdChangeState (eCmdNumber := E_SaMCommandChangeState.Unsuspend);
		E_SaMCommandChangeState.Complete	: THIS^.itfMachineControlHMI.SetCmdChangeState (eCmdNumber := E_SaMCommandChangeState.Complete);
		END_CASE
	END_IF
END_FOR
END_METHOD

(*			
	RafalOS
	Rafał Osajda		24.11.2025		TC 4024.66
	Przygotowanie danych zmiany trybu i jego zmiana
*)
METHOD PRIVATE PrepareChangeMode
VAR_INST
	etmpMode					: E_BaseMachineMode := E_BaseMachineMode.NotAllowed;
END_VAR

VAR
	iJ							: INT;
	iActiveMode					: E_BaseMachineMode;
	etmpCmdChangeMode			: E_SaMCommandChangeMode;
END_VAR
	(*	Przygotowanie ifnormacji dla zmiany trybu	*)

IF (THIS^.refstHMICommonData.bChangePage OR etmpMode <> THIS^.refstData.eActualMode) THEN
	etmpMode := THIS^.refstData.eActualMode;
	THIS^.refstData.iNumberModeToDisplay := 0;
	iActiveMode := THIS^.itfMachineControlHMI.GetActiveMode ();
	FOR iJ := 1 TO GVL_SaMConstans.NUMBER_OF_MODES DO
		IF (THIS^.itfMachineControlHMI.IsModeEnabled (iMode := iJ) AND iJ <> iActiveMode) THEN
			THIS^.refstData.arrNamesOfMode [THIS^.refstData.iNumberModeToDisplay].wsDescription := 
				THIS^.GetTextFromLabelForActiveLocation (stLabel := THIS^.itfMachineControlHMI.GetModeName (iMode := iJ));
			THIS^.refstData.arrNamesOfMode [THIS^.refstData.iNumberModeToDisplay].iNumber := iJ;
			THIS^.refstData.iNumberModeToDisplay := THIS^.refstData.iNumberModeToDisplay + 1;
			THIS^.refstData.iSelectedMode := -1;
		END_IF
	END_FOR
END_IF
IF (THIS^.refstData.bChangeMode AND THIS^.refstData.bSelectedRow) THEN
	THIS^.refstData.bChangeMode := FALSE;
	//polecenie zmiany trybu 
	CASE THIS^.refstData.arrNamesOfMode [THIS^.refstData.iSelectedMode].iNumber OF
	E_SaMCommandChangeMode.Production : etmpCmdChangeMode := E_SaMCommandChangeMode.Production;
	E_SaMCommandChangeMode.Maintenance : etmpCmdChangeMode := E_SaMCommandChangeMode.Maintenance;
	E_SaMCommandChangeMode.Manual : etmpCmdChangeMode := E_SaMCommandChangeMode.Manual;
	E_SaMCommandChangeMode.Washing : etmpCmdChangeMode := E_SaMCommandChangeMode.Washing;
	E_SaMCommandChangeMode.Diagnostisc : etmpCmdChangeMode := E_SaMCommandChangeMode.Diagnostisc;
	END_CASE
	THIS^.itfMachineControlHMI.SetCmdChangeMode (eCmdNumber := etmpCmdChangeMode);
	THIS^.refstData.iSelectedMode := -1;
END_IF
END_METHOD

(*			
	RafalOS
	Rafał Osajda		14.11.2025		TC 4024.66
	Metoda przygotowywania danych dla HMI 
	W niej odbywa się odpytywanie właściego elementu przez łącznik
*)
METHOD PUBLIC PrepareDataForHMI : BOOL
THIS^.refstData.wsActualMode := THIS^.GetTextFromLabelForActiveLocation (THIS^.itfMachineControlHMI.GetActiveModeName ());
THIS^.refstData.eActualMode := THIS^.itfMachineControlHMI.GetActiveMode ();
THIS^.refstData.wsActualState := THIS^.GetTextFromLabelForActiveLocation (THIS^.itfMachineControlHMI.GetActiveStateName ());
THIS^.eActiveMode := THIS^.itfMachineControlHMI.GetActiveMode ();//pobiera numer aktywnego trybu
THIS^.refstData.sTotalWorkTime := THIS^.refstCommonData.itfTime.BaseLTimeToString (
									ltTime 	:= THIS^.itfMachineControlHMI.GetTotalWorkTime (),
									bShowMS	:= FALSE
								);

	(*	Wyświetlenie informacji o stanach pracy				*)

THIS^.PrepareStateInfo ();

	(*	Obsługa przycisków zmiany stanów	*)
	
THIS^.PrepareButtonChangeState ();

	(*	Obsługa zmieny trybów pracy	*)
	
THIS^.PrepareChangeMode ();

	(*	Obsługa informacji zwiazanej z czasami pracy stanach i trybach	*)

IF (THIS^.refstData.bShowTime) THEN
	THIS^.PrepareTimeInfo ();
END_IF

	(*	Obsługa zewnętrzna wyświetlania danych	*)
SUPER^.PrepareDataForHMI ();
END_METHOD

(*			
	RafalOS
	Rafał Osajda		19.11.2025		TC 4024.66
	Przygotowanie ramki pood tamke do wyświetlenia - tylko przygotowanie a nie przygotowanie danych do wyświetlenia
*)
METHOD PUBLIC PrepareForScreen : BOOL
VAR_INPUT
END_VAR
SUPER^.PrepareForScreen ();
END_METHOD

(*			
	RafalOS
	Rafał Osajda		24.11.2025		TC 4024.66
	Wyświetlanie inforamcji o stanach
*)
METHOD PRIVATE PrepareStateInfo
VAR 
	iJ		: INT;
END_VAR
FOR iJ := 0 TO GVL_SaMConstans.NUMBER_OF_STATES DO
	IF (THIS^.itfMachineControlHMI.IsStateEnableInMode (iTestState := iJ)) THEN
		THIS^.refstData.arrStateEnabledInMode [iJ] := TRUE;
	ELSE
		THIS^.refstData.arrStateEnabledInMode [iJ] := FALSE;
	END_IF
	IF (THIS^.itfMachineControlHMI.IsStateActive (iTestState := iJ)) THEN
		THIS^.refstData.arrState [iJ].iWidthFrame := 3;
	ELSE
		THIS^.refstData.arrState [iJ].iWidthFrame := 1;
	END_IF
	
	THIS^.refstData.arrState [iJ].bShowTime := THIS^.refstData.bShowTime;
	THIS^.refstData.arrState [iJ].wsNameOfState := GetTextFromLabelForActiveLocation (THIS^.itfMachineControlHMI.GetStateName (iNumber := iJ));
	IF (THIS^.refstData.arrState [iJ].bShowTime) THEN
		THIS^.refstData.arrState [iJ].sTime := THIS^.refstCommonData.itfTime.BaseLTimeToString (
			ltTime := THIS^.itfMachineControlHMI.GetStateTimeForMode (
						iMode := THIS^.refstData.iNumberModeToShowTime,
						iState := iJ
					),
			bShowMS := FALSE
		);
	ELSE	//czasy dla aktualnego trybu
		THIS^.refstData.arrState [iJ].sTime := THIS^.refstCommonData.itfTime.BaseLTimeToString (
			ltTime := THIS^.itfMachineControlHMI.GetStateTimeForMode (
						iMode := THIS^.eActiveMode,
						iState := iJ
					),
			bShowMS := FALSE
		);
	END_IF
	CASE iJ OF
		2, 5, 7, 11, 14, 17					: THIS^.refstData.arrState [iJ].dwBackgroud := 16#FFDAA520;
		1, 3, 4, 6, 8, 10, 12, 13, 15, 16	: THIS^.refstData.arrState [iJ].dwBackgroud := 16#FF6B8E23;
		9									: THIS^.refstData.arrState [iJ].dwBackgroud := 16#FF00BFFF;
	END_CASE
END_FOR
END_METHOD

(*			
	RafalOS
	Rafał Osajda		24.11.2025		TC 4024.66
	Przygotowanie informacji o czasie pracy w stanie i trybie
*)
METHOD PRIVATE PrepareTimeInfo
VAR_INST
	rtTimeShow					: R_TRIG;
	etmpMode					: E_BaseMachineMode := E_BaseMachineMode.NotAllowed;
END_VAR

	(*	uruchomienie pokazywania danych	*)

rtTimeShow (CLK := THIS^.refstData.bShowTime);
IF (THIS^.refstHMICommonData.bChangePage OR 
		etmpMode <> THIS^.refstData.eActualMode OR 
		rtTimeShow.Q) THEN
	etmpMode := THIS^.refstData.eActualMode;
	THIS^.refstData.iNumberModeToShowTime := THIS^.refstData.eActualMode;
END_IF

	(*	Wartosc dla wyświetlania czasu dla wybranego trybu czasu 	*)

THIS^.refstData.sWorkingTimeInMode := THIS^.refstCommonData.itfTime.BaseLTimeToString (
										ltTime 	:= THIS^.itfMachineControlHMI.GetTimeWorkForMode (
														iMode := THIS^.refstData.iNumberModeToShowTime
													),
										bShowMS	:= FALSE
									);

	(*	Obsługa zmiany trybu dla wyświetlania czasu pracy 	*)

IF (THIS^.refstData.bNextModeToDisplayTime) THEN
	THIS^.refstData.bNextModeToDisplayTime := FALSE;
	REPEAT
		IF (THIS^.refstData.iNumberModeToShowTime + 1 <= GVL_SaMConstans.NUMBER_OF_MODES) THEN
			THIS^.refstData.iNumberModeToShowTime := THIS^.refstData.iNumberModeToShowTime + 1;
		ELSE
			THIS^.refstData.iNumberModeToShowTime := 1;
		END_IF
	UNTIL 
		THIS^.itfMachineControlHMI.IsModeEnabled (iMode := THIS^.refstData.iNumberModeToShowTime)
	END_REPEAT
END_IF
IF (THIS^.refstData.bPrevModeToDisplayTime) THEN
	THIS^.refstData.bPrevModeToDisplayTime := FALSE;
	REPEAT
		IF (THIS^.refstData.iNumberModeToShowTime - 1 >= 1) THEN
			THIS^.refstData.iNumberModeToShowTime := THIS^.refstData.iNumberModeToShowTime - 1;
		ELSE
			THIS^.refstData.iNumberModeToShowTime := GVL_SaMConstans.NUMBER_OF_MODES;
		END_IF
	UNTIL 
		THIS^.itfMachineControlHMI.IsModeEnabled (iMode := THIS^.refstData.iNumberModeToShowTime)
	END_REPEAT
END_IF
THIS^.refstData.wsNameModeOfTimeDisplay := THIS^.GetTextFromLabelForActiveLocation (
											 THIS^.itfMachineControlHMI.GetModeName (iMode := THIS^.refstData.iNumberModeToShowTime)
										);
END_METHOD

END_FUNCTION_BLOCK

// ---- POUs/14_Setings/FB_MCHMIPrepareDataForScreen_07_XX.TcPOU
(*			
	RafalOS
	Rafał Osajda		20.11.2025		TC 4024.66
	Moduł przygotowania danych dla Okna ustawień we wszystkich trybach
*)
FUNCTION_BLOCK FB_MCHMIPrepareDataForScreen_07_XX EXTENDS FB_MCHMIPrepareDataForScreen IMPLEMENTS ITF_MCHMIPrepareDataForScreen
VAR
	itfMachineControlHMI	: ITF_MCHMIMachineControl_HMI_PrepScr_07_XX;
	refstData				: REFERENCE TO ST_MCHMIPrepareScreen_07_XX;
END_VAR

(*			
	RafalOS
	Rafał Osajda		19.11.2025		TC 4024.66
	Czyści danych przy zmienia ramki po poprzedniej ramce
*)
METHOD PUBLIC ClearAfterScreen : BOOL
VAR_INPUT
END_VAR
SUPER^.ClearAfterScreen ();
END_METHOD

METHOD PUBLIC LinkDataHMI_07_XX : BOOL
VAR_INPUT
	refstData				: REFERENCE TO ST_MCHMIPrepareScreen_07_XX;
END_VAR
THIS^.refstData REF= refstData;
END_METHOD

METHOD PUBLIC LinkMachineControlHMI : BOOL
VAR_INPUT
	fbMachineControlHMI	: ITF_MCHMIMachineControl_HMI_PrepScr_07_XX;
END_VAR
this^.itfMachineControlHMI := fbMachineControlHMI;
END_METHOD

(*			
	RafalOS
	Rafał Osajda		14.11.2025		TC 4024.66
	Metoda przygotowywania danych dla HMI 
	W niej odbywa się odpytywanie właściego elementu przez łącznik
*)
METHOD PUBLIC PrepareDataForHMI : BOOL
VAR_INPUT
END_VAR
	(*	Zmiana języka - przygotowanie listy dostępnych języków	*)
THIS^.SettingLocation ();
	
IF (THIS^.refstData.bCreateRecipeTemplate) THEN
	THIS^.refstData.bCreateRecipeTemplate := FALSE;
	THIS^.itfMachineControlHMI.CreateRecipeTemplates ();
END_IF

	(*	Rozszerzenie wyświetlania	*)
SUPER^.PrepareDataForHMI ();
END_METHOD

(*			
	RafalOS
	Rafał Osajda		19.11.2025		TC 4024.66
	Przygotowanie ramki pood tamke do wyświetlenia - tylko przygotowanie a nie przygotowanie danych do wyświetlenia
*)
METHOD PUBLIC PrepareForScreen : BOOL
VAR_INPUT
END_VAR
SUPER^.PrepareForScreen ();
END_METHOD

METHOD PRIVATE SettingLocation : BOOL
VAR_INPUT
END_VAR

VAR
	iI: INT;
	sCodeLocation: STRING;
END_VAR
IF (THIS^.refstHMICommonData.bChangePage) THEN
	FOR iI := 1 TO GVL_BaseConstans.NUMBER_OF_LOCATIONS DO
		THIS^.refstData.arrLocationDescription [iI-1] := THIS^.refstCommonData.itfLocaciotn.GetDescription (iIN := iI);
	END_FOR
	THIS^.refstData.iChoosoLocation := TO_INT (THIS^.refstCommonData.itfLocaciotn.GetLocation ()) - 1;
END_IF

IF ((THIS^.refstData.iChoosoLocation + 1) <> TO_INT (THIS^.refstCommonData.itfLocaciotn.GetLocation ())) THEN
	sCodeLocation := TO_STRING (THIS^.refstCommonData.itfLocaciotn.GetCode (iIN := THIS^.refstData.iChoosoLocation + 1));
	THIS^.refstCommonData.itfLocaciotn.SetLocation (sLocation := TO_STRING (sCodeLocation));
	CURRENTLANGUAGE := sCodeLocation;
END_IF

(*

IF (THIS^.refstOHMI.stUstawienia.iWybranyJezyk <> (TO_INT (THIS^.fbLokalizacja.getJezyk ()) - 1)) THEN
	THIS^.fbLokalizacja.setJezyk (sNowy				:= THIS^.fbLokalizacja.zwrocKod (iIN := THIS^.refstOHMI.stUstawienia.iWybranyJezyk + 1));
	VisuElems.CURRENTLANGUAGE							:= THIS^.fbLokalizacja.zwrocAktualnyKod ();
END_IF
*)
END_METHOD

END_FUNCTION_BLOCK
